LIN {X 0,Y 591.397,Z 324.376,A -85,B 0,C 180,E1 -9125.475,E2 -9125.475} C_VEL
LIN {X 0,Y 591.383,Z 324.375,A -85,B 0,C 180,E1 -9128.017,E2 -9128.017} C_VEL
LIN {X 0,Y 591.414,Z 324.373,A -85,B 0,C 180,E1 -9130.713,E2 -9130.713} C_VEL
LIN {X 0,Y 591.421,Z 324.373,A -85,B 0,C 180,E1 -9133.743,E2 -9133.743} C_VEL
LIN {X 0,Y 591.409,Z 324.376,A -85,B 0,C 180,E1 -9136.612,E2 -9136.612} C_VEL
LIN {X 0,Y 591.432,Z 324.373,A -85,B 0,C 180,E1 -9139.355,E2 -9139.355} C_VEL
LIN {X 0,Y 591.387,Z 324.373,A -85,B 0,C 180,E1 -9141.983,E2 -9141.983} C_VEL
LIN {X 0,Y 591.454,Z 324.372,A -85,B 0,C 180,E1 -9144.529,E2 -9144.529} C_VEL
LIN {X 0,Y 591.403,Z 324.379,A -85,B 0,C 180,E1 -9147.236,E2 -9147.236} C_VEL
LIN {X 0,Y 591.415,Z 324.382,A -85,B 0,C 180,E1 -9149.835,E2 -9149.835} C_VEL
LIN {X 0,Y 591.457,Z 324.484,A -85,B 0,C 180,E1 -9151.821,E2 -9151.821} C_VEL
LIN {X 0,Y 595.055,Z 338.646,A -85,B 0,C 180,E1 -9153.458,E2 -9153.458} C_VEL
LIN {X 0,Y 596.01,Z 344.054,A -85,B 0,C 180,E1 -9154.055,E2 -9154.055} C_VEL
LIN {X 0,Y 595.353,Z 369.323,A -85,B 0,C 180,E1 -9156.59,E2 -9156.59} C_VEL
LIN {X 0,Y 594.51,Z 396.234,A -85,B 0,C 180,E1 -9159.301,E2 -9159.301} C_VEL
LIN {X 0,Y 593.8,Z 422.727,A -85,B 0,C 180,E1 -9161.962,E2 -9161.962} C_VEL
LIN {X 0,Y 593.404,Z 439.816,A -85,B 0,C 180,E1 -9163.676,E2 -9163.676} C_VEL
LIN {X 0,Y 595.77,Z 457.22,A -85,B 0,C 180,E1 -9164.027,E2 -9164.027} C_VEL
LIN {X 0,Y 594.456,Z 560.115,A -85,B 0,C 180,E1 -9165.501,E2 -9165.501} C_VEL
LIN {X 0,Y 594.101,Z 582.366,A -85,B 0,C 180,E1 -9165.839,E2 -9165.839} C_VEL
LIN {X 0,Y 593.767,Z 596.032,A -85,B 0,C 180,E1 -9166.18,E2 -9166.18} C_VEL
LIN {X 0,Y 593.41,Z 609.595,A -85,B 0,C 180,E1 -9166.649,E2 -9166.649} C_VEL
LIN {X 0,Y 592.899,Z 623.687,A -85,B 0,C 180,E1 -9167.289,E2 -9167.289} C_VEL
LIN {X 0,Y 592.458,Z 635.61,A -85,B 0,C 180,E1 -9167.973,E2 -9167.973} C_VEL
LIN {X 0,Y 592.066,Z 646.637,A -85,B 0,C 180,E1 -9168.744,E2 -9168.744} C_VEL
LIN {X 0,Y 591.674,Z 657.474,A -85,B 0,C 180,E1 -9169.656,E2 -9169.656} C_VEL
LIN {X 0,Y 591.308,Z 667.035,A -85,B 0,C 180,E1 -9170.626,E2 -9170.626} C_VEL
LIN {X 0,Y 590.979,Z 675.465,A -85,B 0,C 180,E1 -9171.652,E2 -9171.652} C_VEL
LIN {X 0,Y 590.721,Z 683.499,A -85,B 0,C 180,E1 -9172.848,E2 -9172.848} C_VEL
LIN {X 0,Y 590.563,Z 689.147,A -85,B 0,C 180,E1 -9173.872,E2 -9173.872} C_VEL
LIN {X 0,Y 590.376,Z 695.034,A -85,B 0,C 180,E1 -9175.236,E2 -9175.236} C_VEL
LIN {X 0,Y 590.346,Z 699.319,A -85,B 0,C 180,E1 -9176.599,E2 -9176.599} C_VEL
LIN {X 0,Y 590.252,Z 702.124,A -85,B 0,C 180,E1 -9177.96,E2 -9177.96} C_VEL
LIN {X 0,Y 590.247,Z 703.522,A -85,B 0,C 180,E1 -9179.32,E2 -9179.32} C_VEL
LIN {X 0,Y 590.246,Z 703.516,A -85,B 0,C 180,E1 -9180.68,E2 -9180.68} C_VEL
LIN {X 0,Y 590.25,Z 702.107,A -85,B 0,C 180,E1 -9182.04,E2 -9182.04} C_VEL
LIN {X 0,Y 590.344,Z 699.294,A -85,B 0,C 180,E1 -9183.401,E2 -9183.401} C_VEL
LIN {X 0,Y 590.414,Z 695.001,A -85,B 0,C 180,E1 -9184.764,E2 -9184.764} C_VEL
LIN {X 0,Y 590.509,Z 689.102,A -85,B 0,C 180,E1 -9186.129,E2 -9186.129} C_VEL
LIN {X 0,Y 590.692,Z 682.418,A -85,B 0,C 180,E1 -9187.324,E2 -9187.324} C_VEL
LIN {X 0,Y 590.935,Z 674.066,A -85,B 0,C 180,E1 -9188.521,E2 -9188.521} C_VEL
LIN {X 0,Y 591.277,Z 665.351,A -85,B 0,C 180,E1 -9189.547,E2 -9189.547} C_VEL
LIN {X 0,Y 591.649,Z 654.979,A -85,B 0,C 180,E1 -9190.558,E2 -9190.558} C_VEL
LIN {X 0,Y 591.972,Z 644.168,A -85,B 0,C 180,E1 -9191.431,E2 -9191.431} C_VEL
LIN {X 0,Y 592.438,Z 632.612,A -85,B 0,C 180,E1 -9192.201,E2 -9192.201} C_VEL
LIN {X 0,Y 592.904,Z 619.997,A -85,B 0,C 180,E1 -9192.885,E2 -9192.885} C_VEL
LIN {X 0,Y 593.321,Z 607.005,A -85,B 0,C 180,E1 -9193.44,E2 -9193.44} C_VEL
LIN {X 0,Y 593.593,Z 593.037,A -85,B 0,C 180,E1 -9193.89,E2 -9193.89} C_VEL
LIN {X 0,Y 593.869,Z 578.644,A -85,B 0,C 180,E1 -9194.21,E2 -9194.21} C_VEL
LIN {X 0,Y 595.053,Z 455.793,A -85,B 0,C 180,E1 -9195.884,E2 -9195.884} C_VEL
LIN {X 0,Y 592.977,Z 439.459,A -85,B 0,C 180,E1 -9196.183,E2 -9196.183} C_VEL
LIN {X 0,Y 593.75,Z 410.791,A -85,B 0,C 180,E1 -9199.109,E2 -9199.109} C_VEL
LIN {X 0,Y 594.617,Z 381.153,A -85,B 0,C 180,E1 -9202.145,E2 -9202.145} C_VEL
LIN {X 0,Y 595.362,Z 356.403,A -85,B 0,C 180,E1 -9204.687,E2 -9204.687} C_VEL
LIN {X 0,Y 595.7,Z 344.018,A -85,B 0,C 180,E1 -9205.968,E2 -9205.968} C_VEL
LIN {X 0,Y 592.914,Z 330.893,A -85,B 0,C 180,E1 -9207.435,E2 -9207.435} C_VEL
LIN {X 0,Y 591.482,Z 324.367,A -85,B 0,C 180,E1 -9208.178,E2 -9208.178} C_VEL
LIN {X 0,Y 591.442,Z 324.368,A -85,B 0,C 180,E1 -9210.614,E2 -9210.614} C_VEL
LIN {X 0,Y 591.441,Z 324.372,A -85,B 0,C 180,E1 -9213.01,E2 -9213.01} C_VEL
LIN {X 0,Y 591.491,Z 324.365,A -85,B 0,C 180,E1 -9215.469,E2 -9215.469} C_VEL
LIN {X 0,Y 591.422,Z 324.368,A -85,B 0,C 180,E1 -9218.015,E2 -9218.015} C_VEL
LIN {X 0,Y 591.449,Z 324.368,A -85,B 0,C 180,E1 -9220.717,E2 -9220.717} C_VEL
LIN {X 0,Y 591.424,Z 324.371,A -85,B 0,C 180,E1 -9223.387,E2 -9223.387} C_VEL
LIN {X 0,Y 591.435,Z 324.367,A -85,B 0,C 180,E1 -9226.256,E2 -9226.256} C_VEL
LIN {X 0,Y 591.439,Z 324.37,A -85,B 0,C 180,E1 -9228.455,E2 -9228.455} C_VEL
LIN {X 0,Y 591.415,Z 324.372,A -85,B 0,C 180,E1 -9231.119,E2 -9231.119} C_VEL
LIN {X 0,Y 591.426,Z 324.37,A -85,B 0,C 180,E1 -9232.22,E2 -9232.22} C_VEL
LIN {X 0,Y 590.787,Z 324.455,A -85,B 0,C 180,E1 -9232.788,E2 -9232.788} C_VEL
LIN {X 0,Y 587.96,Z 324.808,A -85,B 0,C 180,E1 -9233.711,E2 -9233.711} C_VEL
LIN {X 0,Y 585.55,Z 325.106,A -85,B 0,C 180,E1 -9234.454,E2 -9234.454} C_VEL
LIN {X 0,Y 584.503,Z 325.233,A -85,B 0,C 180,E1 -9235.027,E2 -9235.027} C_VEL
LIN {X 0,Y 584.412,Z 325.242,A -85,B 0,C 180,E1 -9235.221,E2 -9235.221} C_VEL
LIN {X 0,Y 584.395,Z 325.248,A -85,B 0,C 180,E1 -9238.172,E2 -9238.172} C_VEL
LIN {X 0,Y 584.426,Z 325.241,A -85,B 0,C 180,E1 -9241.036,E2 -9241.036} C_VEL
LIN {X 0,Y 584.36,Z 325.249,A -85,B 0,C 180,E1 -9243.673,E2 -9243.673} C_VEL
LIN {X 0,Y 584.413,Z 325.246,A -85,B 0,C 180,E1 -9245.952,E2 -9245.952} C_VEL
LIN {X 0,Y 584.451,Z 325.237,A -85,B 0,C 180,E1 -9248.928,E2 -9248.928} C_VEL
LIN {X 0,Y 584.403,Z 325.249,A -85,B 0,C 180,E1 -9251.843,E2 -9251.843} C_VEL
LIN {X 0,Y 584.433,Z 325.24,A -85,B 0,C 180,E1 -9254.712,E2 -9254.712} C_VEL
LIN {X 0,Y 584.455,Z 325.237,A -85,B 0,C 180,E1 -9256.838,E2 -9256.838} C_VEL
LIN {X 0,Y 584.458,Z 325.239,A -85,B 0,C 180,E1 -9258.945,E2 -9258.945} C_VEL
LIN {X 0,Y 588.396,Z 337.126,A -85,B 0,C 180,E1 -9259.205,E2 -9259.205} C_VEL
LIN {X 0,Y 587.901,Z 445.913,A -85,B 0,C 180,E1 -9260.55,E2 -9260.55} C_VEL
LIN {X 0,Y 587.79,Z 460.378,A -85,B 0,C 180,E1 -9260.851,E2 -9260.851} C_VEL
LIN {X 0,Y 587.602,Z 473.525,A -85,B 0,C 180,E1 -9261.258,E2 -9261.258} C_VEL
LIN {X 0,Y 587.302,Z 485.998,A -85,B 0,C 180,E1 -9261.772,E2 -9261.772} C_VEL
LIN {X 0,Y 586.938,Z 498.954,A -85,B 0,C 180,E1 -9262.457,E2 -9262.457} C_VEL
LIN {X 0,Y 586.539,Z 510.662,A -85,B 0,C 180,E1 -9263.228,E2 -9263.228} C_VEL
LIN {X 0,Y 586.082,Z 520.417,A -85,B 0,C 180,E1 -9263.997,E2 -9263.997} C_VEL
LIN {X 0,Y 585.592,Z 531.141,A -85,B 0,C 180,E1 -9265.025,E2 -9265.025} C_VEL
LIN {X 0,Y 585.201,Z 540,A -85,B 0,C 180,E1 -9266.054,E2 -9266.054} C_VEL
LIN {X 0,Y 584.818,Z 548.476,A -85,B 0,C 180,E1 -9267.254,E2 -9267.254} C_VEL
LIN {X 0,Y 584.51,Z 554.451,A -85,B 0,C 180,E1 -9268.283,E2 -9268.283} C_VEL
LIN {X 0,Y 584.27,Z 559.407,A -85,B 0,C 180,E1 -9269.313,E2 -9269.313} C_VEL
LIN {X 0,Y 583.986,Z 564.529,A -85,B 0,C 180,E1 -9270.687,E2 -9270.687} C_VEL
LIN {X 0,Y 583.898,Z 568.164,A -85,B 0,C 180,E1 -9272.063,E2 -9272.063} C_VEL
LIN {X 0,Y 583.945,Z 570.435,A -85,B 0,C 180,E1 -9273.439,E2 -9273.439} C_VEL
LIN {X 0,Y 583.832,Z 571.428,A -85,B 0,C 180,E1 -9274.818,E2 -9274.818} C_VEL
LIN {X 0,Y 583.931,Z 571.112,A -85,B 0,C 180,E1 -9276.198,E2 -9276.198} C_VEL
LIN {X 0,Y 584.001,Z 569.505,A -85,B 0,C 180,E1 -9277.581,E2 -9277.581} C_VEL
LIN {X 0,Y 584.104,Z 566.555,A -85,B 0,C 180,E1 -9278.969,E2 -9278.969} C_VEL
LIN {X 0,Y 584.448,Z 562.149,A -85,B 0,C 180,E1 -9280.357,E2 -9280.357} C_VEL
LIN {X 0,Y 584.647,Z 557.768,A -85,B 0,C 180,E1 -9281.402,E2 -9281.402} C_VEL
LIN {X 0,Y 584.964,Z 552.416,A -85,B 0,C 180,E1 -9282.447,E2 -9282.447} C_VEL
LIN {X 0,Y 585.399,Z 544.728,A -85,B 0,C 180,E1 -9283.669,E2 -9283.669} C_VEL
LIN {X 0,Y 585.867,Z 536.664,A -85,B 0,C 180,E1 -9284.718,E2 -9284.718} C_VEL
LIN {X 0,Y 586.358,Z 526.909,A -85,B 0,C 180,E1 -9285.769,E2 -9285.769} C_VEL
LIN {X 0,Y 586.796,Z 517.087,A -85,B 0,C 180,E1 -9286.648,E2 -9286.648} C_VEL
LIN {X 0,Y 587.203,Z 506.593,A -85,B 0,C 180,E1 -9287.431,E2 -9287.431} C_VEL
LIN {X 0,Y 587.739,Z 494.971,A -85,B 0,C 180,E1 -9288.141,E2 -9288.141} C_VEL
LIN {X 0,Y 588.097,Z 482.425,A -85,B 0,C 180,E1 -9288.759,E2 -9288.759} C_VEL
LIN {X 0,Y 588.319,Z 469.674,A -85,B 0,C 180,E1 -9289.247,E2 -9289.247} C_VEL
LIN {X 0,Y 588.494,Z 455.956,A -85,B 0,C 180,E1 -9289.631,E2 -9289.631} C_VEL
LIN {X 0,Y 588.639,Z 442.281,A -85,B 0,C 180,E1 -9289.877,E2 -9289.877} C_VEL
LIN {X 0,Y 589.266,Z 338.454,A -85,B 0,C 180,E1 -9291.162,E2 -9291.162} C_VEL
LIN {X 0,Y 584.397,Z 325.318,A -85,B 0,C 180,E1 -9291.488,E2 -9291.488} C_VEL
LIN {X 0,Y 584.399,Z 325.253,A -85,B 0,C 180,E1 -9294.367,E2 -9294.367} C_VEL
LIN {X 0,Y 584.392,Z 325.248,A -85,B 0,C 180,E1 -9297.506,E2 -9297.506} C_VEL
LIN {X 0,Y 584.358,Z 325.257,A -85,B 0,C 180,E1 -9300.341,E2 -9300.341} C_VEL
LIN {X 0,Y 584.359,Z 325.25,A -85,B 0,C 180,E1 -9302.959,E2 -9302.959} C_VEL
LIN {X 0,Y 584.365,Z 325.253,A -85,B 0,C 180,E1 -9305.968,E2 -9305.968} C_VEL
LIN {X 0,Y 584.364,Z 325.249,A -85,B 0,C 180,E1 -9308.819,E2 -9308.819} C_VEL
LIN {X 0,Y 584.345,Z 325.251,A -85,B 0,C 180,E1 -9311.245,E2 -9311.245} C_VEL
LIN {X 0,Y 584.397,Z 325.252,A -85,B 0,C 180,E1 -9314.042,E2 -9314.042} C_VEL
LIN {X 0,Y 584.394,Z 325.244,A -85,B 0,C 180,E1 -9316.982,E2 -9316.982} C_VEL
LIN {X 0,Y 584.359,Z 325.253,A -85,B 0,C 180,E1 -9320.098,E2 -9320.098} C_VEL
LIN {X 0,Y 584.342,Z 325.238,A -85,B 0,C 180,E1 -9322.314,E2 -9322.314} C_VEL
LIN {X 0,Y 584.353,Z 325.24,A -85,B 0,C 180,E1 -9324.875,E2 -9324.875} C_VEL
LIN {X 0,Y 584.358,Z 325.249,A -85,B 0,C 180,E1 -9327.357,E2 -9327.357} C_VEL
LIN {X 0,Y 584.371,Z 325.248,A -85,B 0,C 180,E1 -9329.773,E2 -9329.773} C_VEL
LIN {X 0,Y 584.392,Z 325.242,A -85,B 0,C 180,E1 -9332.494,E2 -9332.494} C_VEL
LIN {X 0,Y 584.399,Z 325.248,A -85,B 0,C 180,E1 -9335.633,E2 -9335.633} C_VEL
LIN {X 0,Y 584.372,Z 325.244,A -85,B 0,C 180,E1 -9338.187,E2 -9338.187} C_VEL
LIN {X 0,Y 584.372,Z 325.25,A -85,B 0,C 180,E1 -9340.39,E2 -9340.39} C_VEL
LIN {X 0,Y 584.408,Z 325.251,A -85,B 0,C 180,E1 -9343.08,E2 -9343.08} C_VEL
LIN {X 0,Y 588.095,Z 337.425,A -85,B 0,C 180,E1 -9343.346,E2 -9343.346} C_VEL
LIN {X 0,Y 587.069,Z 446.386,A -85,B 0,C 180,E1 -9344.858,E2 -9344.858} C_VEL
LIN {X 0,Y 586.891,Z 461.083,A -85,B 0,C 180,E1 -9345.208,E2 -9345.208} C_VEL
LIN {X 0,Y 586.707,Z 475.547,A -85,B 0,C 180,E1 -9345.701,E2 -9345.701} C_VEL
LIN {X 0,Y 586.399,Z 488.186,A -85,B 0,C 180,E1 -9346.266,E2 -9346.266} C_VEL
LIN {X 0,Y 586.061,Z 500.538,A -85,B 0,C 180,E1 -9346.962,E2 -9346.962} C_VEL
LIN {X 0,Y 585.664,Z 512.992,A -85,B 0,C 180,E1 -9347.831,E2 -9347.831} C_VEL
LIN {X 0,Y 585.28,Z 524.558,A -85,B 0,C 180,E1 -9348.819,E2 -9348.819} C_VEL
LIN {X 0,Y 585.02,Z 534.267,A -85,B 0,C 180,E1 -9349.828,E2 -9349.828} C_VEL
LIN {X 0,Y 584.669,Z 542.575,A -85,B 0,C 180,E1 -9350.866,E2 -9350.866} C_VEL
LIN {X 0,Y 584.376,Z 550.49,A -85,B 0,C 180,E1 -9352.077,E2 -9352.077} C_VEL
LIN {X 0,Y 584.167,Z 556.045,A -85,B 0,C 180,E1 -9353.113,E2 -9353.113} C_VEL
LIN {X 0,Y 583.969,Z 561.848,A -85,B 0,C 180,E1 -9354.493,E2 -9354.493} C_VEL
LIN {X 0,Y 583.887,Z 566.071,A -85,B 0,C 180,E1 -9355.872,E2 -9355.872} C_VEL
LIN {X 0,Y 583.89,Z 568.829,A -85,B 0,C 180,E1 -9357.249,E2 -9357.249} C_VEL
LIN {X 0,Y 583.722,Z 570.182,A -85,B 0,C 180,E1 -9358.625,E2 -9358.625} C_VEL
LIN {X 0,Y 583.655,Z 570.168,A -85,B 0,C 180,E1 -9360,E2 -9360} C_VEL
LIN {X 0,Y 583.751,Z 568.777,A -85,B 0,C 180,E1 -9361.375,E2 -9361.375} C_VEL
LIN {X 0,Y 584.059,Z 565.978,A -85,B 0,C 180,E1 -9362.749,E2 -9362.749} C_VEL
LIN {X 0,Y 584.433,Z 561.687,A -85,B 0,C 180,E1 -9364.124,E2 -9364.124} C_VEL
LIN {X 0,Y 584.407,Z 555.792,A -85,B 0,C 180,E1 -9365.502,E2 -9365.502} C_VEL
LIN {X 0,Y 584.916,Z 549.091,A -85,B 0,C 180,E1 -9366.705,E2 -9366.705} C_VEL
LIN {X 0,Y 585.301,Z 540.781,A -85,B 0,C 180,E1 -9367.91,E2 -9367.91} C_VEL
LIN {X 0,Y 585.641,Z 532.032,A -85,B 0,C 180,E1 -9368.945,E2 -9368.945} C_VEL
LIN {X 0,Y 586.047,Z 521.342,A -85,B 0,C 180,E1 -9369.98,E2 -9369.98} C_VEL
LIN {X 0,Y 586.402,Z 512.877,A -85,B 0,C 180,E1 -9370.669,E2 -9370.669} C_VEL
LIN {X 0,Y 586.82,Z 501.498,A -85,B 0,C 180,E1 -9371.446,E2 -9371.446} C_VEL
LIN {X 0,Y 587.254,Z 488.639,A -85,B 0,C 180,E1 -9372.154,E2 -9372.154} C_VEL
LIN {X 0,Y 587.518,Z 475.083,A -85,B 0,C 180,E1 -9372.742,E2 -9372.742} C_VEL
LIN {X 0,Y 587.697,Z 460.944,A -85,B 0,C 180,E1 -9373.198,E2 -9373.198} C_VEL
LIN {X 0,Y 587.824,Z 446.981,A -85,B 0,C 180,E1 -9373.502,E2 -9373.502} C_VEL
LIN {X 0,Y 589.193,Z 337.801,A -85,B 0,C 180,E1 -9375.112,E2 -9375.112} C_VEL
LIN {X 0,Y 584.475,Z 325.436,A -85,B 0,C 180,E1 -9375.495,E2 -9375.495} C_VEL
LIN {X 0,Y 584.403,Z 325.252,A -85,B 0,C 180,E1 -9378.157,E2 -9378.157} C_VEL
LIN {X 0,Y 584.45,Z 325.241,A -85,B 0,C 180,E1 -9381.072,E2 -9381.072} C_VEL
LIN {X 0,Y 584.432,Z 325.249,A -85,B 0,C 180,E1 -9384.047,E2 -9384.047} C_VEL
LIN {X 0,Y 584.375,Z 325.25,A -85,B 0,C 180,E1 -9387.095,E2 -9387.095} C_VEL
LIN {X 0,Y 584.406,Z 325.247,A -85,B 0,C 180,E1 -9389.433,E2 -9389.433} C_VEL
LIN {X 0,Y 584.395,Z 325.249,A -85,B 0,C 180,E1 -9391.828,E2 -9391.828} C_VEL
LIN {X 0,Y 584.405,Z 325.242,A -85,B 0,C 180,E1 -9394.286,E2 -9394.286} C_VEL
LIN {X 0,Y 584.423,Z 325.239,A -85,B 0,C 180,E1 -9396.817,E2 -9396.817} C_VEL
LIN {X 0,Y 584.359,Z 325.246,A -85,B 0,C 180,E1 -9399.902,E2 -9399.902} C_VEL
LIN {X 0,Y 584.393,Z 325.24,A -85,B 0,C 180,E1 -9402.16,E2 -9402.16} C_VEL
LIN {X 0,Y 584.394,Z 325.249,A -85,B 0,C 180,E1 -9405.005,E2 -9405.005} C_VEL
LIN {X 0,Y 584.388,Z 325.244,A -85,B 0,C 180,E1 -9407.999,E2 -9407.999} C_VEL
LIN {X 0,Y 584.352,Z 325.254,A -85,B 0,C 180,E1 -9410.558,E2 -9410.558} C_VEL
LIN {X 0,Y 584.359,Z 325.251,A -85,B 0,C 180,E1 -9413.427,E2 -9413.427} C_VEL
LIN {X 0,Y 584.331,Z 325.249,A -85,B 0,C 180,E1 -9415.803,E2 -9415.803} C_VEL
LIN {X 0,Y 584.383,Z 325.253,A -85,B 0,C 180,E1 -9418.322,E2 -9418.322} C_VEL
LIN {X 0,Y 584.394,Z 325.249,A -85,B 0,C 180,E1 -9421.351,E2 -9421.351} C_VEL
LIN {X 0,Y 584.426,Z 325.373,A -85,B 0,C 180,E1 -9421.646,E2 -9421.646} C_VEL
LIN {X 0,Y 588.255,Z 343.449,A -85,B 0,C 180,E1 -9423.86,E2 -9423.86} C_VEL
LIN {X 0,Y 587.403,Z 365.293,A -85,B 0,C 180,E1 -9426.266,E2 -9426.266} C_VEL
LIN {X 0,Y 586.297,Z 393.805,A -85,B 0,C 180,E1 -9429.364,E2 -9429.364} C_VEL
LIN {X 0,Y 585.464,Z 418.853,A -85,B 0,C 180,E1 -9432.057,E2 -9432.057} C_VEL
LIN {X 0,Y 585.077,Z 431.768,A -85,B 0,C 180,E1 -9433.438,E2 -9433.438} C_VEL
LIN {X 0,Y 588.218,Z 459.236,A -85,B 0,C 180,E1 -9433.885,E2 -9433.885} C_VEL
LIN {X 0,Y 588.563,Z 466.079,A -85,B 0,C 180,E1 -9433.981,E2 -9433.981} C_VEL
LIN {X 0,Y 587.657,Z 571.482,A -85,B 0,C 180,E1 -9435.287,E2 -9435.287} C_VEL
LIN {X 0,Y 587.212,Z 585.956,A -85,B 0,C 180,E1 -9435.603,E2 -9435.603} C_VEL
LIN {X 0,Y 586.633,Z 599.953,A -85,B 0,C 180,E1 -9436.052,E2 -9436.052} C_VEL
LIN {X 0,Y 586.09,Z 613.003,A -85,B 0,C 180,E1 -9436.611,E2 -9436.611} C_VEL
LIN {X 0,Y 585.491,Z 625.675,A -85,B 0,C 180,E1 -9437.301,E2 -9437.301} C_VEL
LIN {X 0,Y 584.924,Z 641.523,A -85,B 0,C 180,E1 -9438.254,E2 -9438.254} C_VEL
LIN {X 0,Y 584.541,Z 653.444,A -85,B 0,C 180,E1 -9439.136,E2 -9439.136} C_VEL
LIN {X 0,Y 584.21,Z 662.96,A -85,B 0,C 180,E1 -9439.988,E2 -9439.988} C_VEL
LIN {X 0,Y 583.917,Z 672.662,A -85,B 0,C 180,E1 -9441.028,E2 -9441.028} C_VEL
LIN {X 0,Y 583.658,Z 681.865,A -85,B 0,C 180,E1 -9442.241,E2 -9442.241} C_VEL
LIN {X 0,Y 583.481,Z 689.238,A -85,B 0,C 180,E1 -9443.451,E2 -9443.451} C_VEL
LIN {X 0,Y 583.422,Z 694.371,A -85,B 0,C 180,E1 -9444.488,E2 -9444.488} C_VEL
LIN {X 0,Y 583.291,Z 699.616,A -85,B 0,C 180,E1 -9445.868,E2 -9445.868} C_VEL
LIN {X 0,Y 583.27,Z 703.288,A -85,B 0,C 180,E1 -9447.247,E2 -9447.247} C_VEL
LIN {X 0,Y 583.251,Z 705.492,A -85,B 0,C 180,E1 -9448.624,E2 -9448.624} C_VEL
LIN {X 0,Y 583.252,Z 706.28,A -85,B 0,C 180,E1 -9450,E2 -9450} C_VEL
LIN {X 0,Y 583.25,Z 705.646,A -85,B 0,C 180,E1 -9451.376,E2 -9451.376} C_VEL
LIN {X 0,Y 583.27,Z 703.57,A -85,B 0,C 180,E1 -9452.753,E2 -9452.753} C_VEL
LIN {X 0,Y 583.308,Z 700.026,A -85,B 0,C 180,E1 -9454.132,E2 -9454.132} C_VEL
LIN {X 0,Y 583.422,Z 694.91,A -85,B 0,C 180,E1 -9455.511,E2 -9455.511} C_VEL
LIN {X 0,Y 583.501,Z 689.927,A -85,B 0,C 180,E1 -9456.548,E2 -9456.548} C_VEL
LIN {X 0,Y 583.682,Z 682.734,A -85,B 0,C 180,E1 -9457.759,E2 -9457.759} C_VEL
LIN {X 0,Y 583.902,Z 675.173,A -85,B 0,C 180,E1 -9458.798,E2 -9458.798} C_VEL
LIN {X 0,Y 584.258,Z 666.053,A -85,B 0,C 180,E1 -9459.836,E2 -9459.836} C_VEL
LIN {X 0,Y 584.613,Z 656.484,A -85,B 0,C 180,E1 -9460.744,E2 -9460.744} C_VEL
LIN {X 0,Y 585.045,Z 644.9,A -85,B 0,C 180,E1 -9461.656,E2 -9461.656} C_VEL
LIN {X 0,Y 585.416,Z 632.766,A -85,B 0,C 180,E1 -9462.437,E2 -9462.437} C_VEL
LIN {X 0,Y 585.937,Z 619.165,A -85,B 0,C 180,E1 -9463.128,E2 -9463.128} C_VEL
LIN {X 0,Y 586.311,Z 604.779,A -85,B 0,C 180,E1 -9463.691,E2 -9463.691} C_VEL
LIN {X 0,Y 586.943,Z 582.569,A -85,B 0,C 180,E1 -9464.315,E2 -9464.315} C_VEL
LIN {X 0,Y 587.347,Z 568.106,A -85,B 0,C 180,E1 -9464.59,E2 -9464.59} C_VEL
LIN {X 0,Y 587.831,Z 505.932,A -85,B 0,C 180,E1 -9465.374,E2 -9465.374} C_VEL
LIN {X 0,Y 588.355,Z 461.363,A -85,B 0,C 180,E1 -9466.058,E2 -9466.058} C_VEL
LIN {X 0,Y 586.017,Z 437.005,A -85,B 0,C 180,E1 -9466.538,E2 -9466.538} C_VEL
LIN {X 0,Y 585.044,Z 427.965,A -85,B 0,C 180,E1 -9466.779,E2 -9466.779} C_VEL
LIN {X 0,Y 585.853,Z 398.261,A -85,B 0,C 180,E1 -9469.922,E2 -9469.922} C_VEL
LIN {X 0,Y 586.666,Z 372.688,A -85,B 0,C 180,E1 -9472.647,E2 -9472.647} C_VEL
LIN {X 0,Y 587.629,Z 345.22,A -85,B 0,C 180,E1 -9475.601,E2 -9475.601} C_VEL
LIN {X 0,Y 587.678,Z 341.765,A -85,B 0,C 180,E1 -9475.977,E2 -9475.977} C_VEL
LIN {X 0,Y 584.405,Z 325.25,A -85,B 0,C 180,E1 -9477.917,E2 -9477.917} C_VEL
LIN {X 0,Y 584.354,Z 325.25,A -85,B 0,C 180,E1 -9480.341,E2 -9480.341} C_VEL
LIN {X 0,Y 584.357,Z 325.251,A -85,B 0,C 180,E1 -9482.959,E2 -9482.959} C_VEL
LIN {X 0,Y 584.346,Z 325.253,A -85,B 0,C 180,E1 -9485.97,E2 -9485.97} C_VEL
LIN {X 0,Y 584.349,Z 325.253,A -85,B 0,C 180,E1 -9488.818,E2 -9488.818} C_VEL
LIN {X 0,Y 584.34,Z 325.254,A -85,B 0,C 180,E1 -9491.245,E2 -9491.245} C_VEL
LIN {X 0,Y 584.392,Z 325.247,A -85,B 0,C 180,E1 -9494.042,E2 -9494.042} C_VEL
LIN {X 0,Y 584.357,Z 325.253,A -85,B 0,C 180,E1 -9496.986,E2 -9496.986} C_VEL
LIN {X 0,Y 584.355,Z 325.251,A -85,B 0,C 180,E1 -9500.098,E2 -9500.098} C_VEL
LIN {X 0,Y 584.371,Z 325.249,A -85,B 0,C 180,E1 -9502.316,E2 -9502.316} C_VEL
LIN {X 0,Y 584.404,Z 325.249,A -85,B 0,C 180,E1 -9504.879,E2 -9504.879} C_VEL
LIN {X 0,Y 584.357,Z 325.258,A -85,B 0,C 180,E1 -9507.358,E2 -9507.358} C_VEL
LIN {X 0,Y 584.377,Z 325.259,A -85,B 0,C 180,E1 -9509.774,E2 -9509.774} C_VEL
LIN {X 0,Y 584.407,Z 325.27,A -85,B 0,C 180,E1 -9511.499,E2 -9511.499} C_VEL
LIN {X 0,Y 588.269,Z 340.159,A -85,B 0,C 180,E1 -9513.255,E2 -9513.255} C_VEL
LIN {X 0,Y 589.318,Z 345.96,A -85,B 0,C 180,E1 -9513.911,E2 -9513.911} C_VEL
LIN {X 0,Y 588.635,Z 370.358,A -85,B 0,C 180,E1 -9516.386,E2 -9516.386} C_VEL
LIN {X 0,Y 587.776,Z 396.637,A -85,B 0,C 180,E1 -9519.053,E2 -9519.053} C_VEL
LIN {X 0,Y 586.971,Z 423.126,A -85,B 0,C 180,E1 -9521.745,E2 -9521.745} C_VEL
LIN {X 0,Y 586.595,Z 439.961,A -85,B 0,C 180,E1 -9523.436,E2 -9523.436} C_VEL
LIN {X 0,Y 589.053,Z 457.646,A -85,B 0,C 180,E1 -9523.807,E2 -9523.807} C_VEL
LIN {X 0,Y 587.618,Z 560.787,A -85,B 0,C 180,E1 -9525.324,E2 -9525.324} C_VEL
LIN {X 0,Y 587.257,Z 581.978,A -85,B 0,C 180,E1 -9525.649,E2 -9525.649} C_VEL
LIN {X 0,Y 586.896,Z 596.435,A -85,B 0,C 180,E1 -9526.015,E2 -9526.015} C_VEL
LIN {X 0,Y 586.517,Z 609.87,A -85,B 0,C 180,E1 -9526.49,E2 -9526.49} C_VEL
LIN {X 0,Y 585.983,Z 623.876,A -85,B 0,C 180,E1 -9527.137,E2 -9527.137} C_VEL
LIN {X 0,Y 585.529,Z 635.745,A -85,B 0,C 180,E1 -9527.829,E2 -9527.829} C_VEL
LIN {X 0,Y 585.08,Z 646.743,A -85,B 0,C 180,E1 -9528.607,E2 -9528.607} C_VEL
LIN {X 0,Y 584.668,Z 657.182,A -85,B 0,C 180,E1 -9529.494,E2 -9529.494} C_VEL
LIN {X 0,Y 584.299,Z 667.131,A -85,B 0,C 180,E1 -9530.513,E2 -9530.513} C_VEL
LIN {X 0,Y 583.94,Z 675.544,A -85,B 0,C 180,E1 -9531.55,E2 -9531.55} C_VEL
LIN {X 0,Y 583.642,Z 683.568,A -85,B 0,C 180,E1 -9532.761,E2 -9532.761} C_VEL
LIN {X 0,Y 583.498,Z 689.205,A -85,B 0,C 180,E1 -9533.798,E2 -9533.798} C_VEL
LIN {X 0,Y 583.291,Z 695.093,A -85,B 0,C 180,E1 -9535.178,E2 -9535.178} C_VEL
LIN {X 0,Y 583.259,Z 699.374,A -85,B 0,C 180,E1 -9536.558,E2 -9536.558} C_VEL
LIN {X 0,Y 583.163,Z 702.17,A -85,B 0,C 180,E1 -9537.935,E2 -9537.935} C_VEL
LIN {X 0,Y 583.147,Z 703.55,A -85,B 0,C 180,E1 -9539.312,E2 -9539.312} C_VEL
LIN {X 0,Y 583.146,Z 703.517,A -85,B 0,C 180,E1 -9540.688,E2 -9540.688} C_VEL
LIN {X 0,Y 583.161,Z 702.083,A -85,B 0,C 180,E1 -9542.065,E2 -9542.065} C_VEL
LIN {X 0,Y 583.255,Z 699.239,A -85,B 0,C 180,E1 -9543.443,E2 -9543.443} C_VEL
LIN {X 0,Y 583.323,Z 694.911,A -85,B 0,C 180,E1 -9544.822,E2 -9544.822} C_VEL
LIN {X 0,Y 583.43,Z 688.966,A -85,B 0,C 180,E1 -9546.203,E2 -9546.203} C_VEL
LIN {X 0,Y 583.634,Z 682.22,A -85,B 0,C 180,E1 -9547.413,E2 -9547.413} C_VEL
LIN {X 0,Y 583.86,Z 673.804,A -85,B 0,C 180,E1 -9548.625,E2 -9548.625} C_VEL
LIN {X 0,Y 584.233,Z 665.021,A -85,B 0,C 180,E1 -9549.663,E2 -9549.663} C_VEL
LIN {X 0,Y 584.591,Z 655.602,A -85,B 0,C 180,E1 -9550.593,E2 -9550.593} C_VEL
LIN {X 0,Y 584.929,Z 644.812,A -85,B 0,C 180,E1 -9551.484,E2 -9551.484} C_VEL
LIN {X 0,Y 585.375,Z 633.371,A -85,B 0,C 180,E1 -9552.263,E2 -9552.263} C_VEL
LIN {X 0,Y 585.861,Z 620.916,A -85,B 0,C 180,E1 -9552.954,E2 -9552.954} C_VEL
LIN {X 0,Y 586.329,Z 607.105,A -85,B 0,C 180,E1 -9553.559,E2 -9553.559} C_VEL
LIN {X 0,Y 586.612,Z 593.187,A -85,B 0,C 180,E1 -9554.015,E2 -9554.015} C_VEL
LIN {X 0,Y 586.918,Z 578.92,A -85,B 0,C 180,E1 -9554.338,E2 -9554.338} C_VEL
LIN {X 0,Y 588.223,Z 456.806,A -85,B 0,C 180,E1 -9556.037,E2 -9556.037} C_VEL
LIN {X 0,Y 586.038,Z 439.461,A -85,B 0,C 180,E1 -9556.357,E2 -9556.357} C_VEL
LIN {X 0,Y 586.876,Z 409.273,A -85,B 0,C 180,E1 -9559.459,E2 -9559.459} C_VEL
LIN {X 0,Y 587.74,Z 380.6,A -85,B 0,C 180,E1 -9562.418,E2 -9562.418} C_VEL
LIN {X 0,Y 588.606,Z 354.291,A -85,B 0,C 180,E1 -9565.147,E2 -9565.147} C_VEL
LIN {X 0,Y 588.763,Z 344.951,A -85,B 0,C 180,E1 -9566.116,E2 -9566.116} C_VEL
LIN {X 0,Y 584.447,Z 325.243,A -85,B 0,C 180,E1 -9568.377,E2 -9568.377} C_VEL
LIN {X 0,Y 584.406,Z 325.248,A -85,B 0,C 180,E1 -9571.023,E2 -9571.023} C_VEL
LIN {X 0,Y 584.388,Z 325.251,A -85,B 0,C 180,E1 -9573.46,E2 -9573.46} C_VEL
LIN {X 0,Y 584.428,Z 325.239,A -85,B 0,C 180,E1 -9575.964,E2 -9575.964} C_VEL
LIN {X 0,Y 584.368,Z 325.251,A -85,B 0,C 180,E1 -9578.82,E2 -9578.82} C_VEL
LIN {X 0,Y 584.384,Z 325.25,A -85,B 0,C 180,E1 -9581.242,E2 -9581.242} C_VEL
LIN {X 0,Y 584.398,Z 325.243,A -85,B 0,C 180,E1 -9584.041,E2 -9584.041} C_VEL
LIN {X 0,Y 584.401,Z 325.25,A -85,B 0,C 180,E1 -9586.981,E2 -9586.981} C_VEL
LIN {X 0,Y 584.415,Z 325.241,A -85,B 0,C 180,E1 -9589.668,E2 -9589.668} C_VEL
LIN {X 0,Y 584.386,Z 325.248,A -85,B 0,C 180,E1 -9592.317,E2 -9592.317} C_VEL
LIN {X 0,Y 584.441,Z 325.242,A -85,B 0,C 180,E1 -9594.881,E2 -9594.881} C_VEL
LIN {X 0,Y 584.412,Z 325.242,A -85,B 0,C 180,E1 -9595.221,E2 -9595.221} C_VEL
LIN {X 0,Y 583.729,Z 325.327,A -85,B 0,C 180,E1 -9595.796,E2 -9595.796} C_VEL
LIN {X 0,Y 580.87,Z 325.688,A -85,B 0,C 180,E1 -9596.729,E2 -9596.729} C_VEL
LIN {X 0,Y 578.462,Z 325.986,A -85,B 0,C 180,E1 -9597.479,E2 -9597.479} C_VEL
LIN {X 0,Y 577.428,Z 326.115,A -85,B 0,C 180,E1 -9598.059,E2 -9598.059} C_VEL
LIN {X 0,Y 577.343,Z 326.126,A -85,B 0,C 180,E1 -9598.255,E2 -9598.255} C_VEL
LIN {X 0,Y 577.391,Z 326.117,A -85,B 0,C 180,E1 -9600.971,E2 -9600.971} C_VEL
LIN {X 0,Y 577.316,Z 326.128,A -85,B 0,C 180,E1 -9603.874,E2 -9603.874} C_VEL
LIN {X 0,Y 577.359,Z 326.126,A -85,B 0,C 180,E1 -9606.4,E2 -9606.4} C_VEL
LIN {X 0,Y 577.399,Z 326.116,A -85,B 0,C 180,E1 -9609.082,E2 -9609.082} C_VEL
LIN {X 0,Y 577.383,Z 326.12,A -85,B 0,C 180,E1 -9611.614,E2 -9611.614} C_VEL
LIN {X 0,Y 577.399,Z 326.117,A -85,B 0,C 180,E1 -9614.521,E2 -9614.521} C_VEL
LIN {X 0,Y 577.41,Z 326.114,A -85,B 0,C 180,E1 -9616.674,E2 -9616.674} C_VEL
LIN {X 0,Y 577.421,Z 326.115,A -85,B 0,C 180,E1 -9618.764,E2 -9618.764} C_VEL
LIN {X 0,Y 581.561,Z 338.528,A -85,B 0,C 180,E1 -9619.041,E2 -9619.041} C_VEL
LIN {X 0,Y 581.028,Z 446.658,A -85,B 0,C 180,E1 -9620.393,E2 -9620.393} C_VEL
LIN {X 0,Y 580.908,Z 461.132,A -85,B 0,C 180,E1 -9620.697,E2 -9620.697} C_VEL
LIN {X 0,Y 580.698,Z 474.286,A -85,B 0,C 180,E1 -9621.11,E2 -9621.11} C_VEL
LIN {X 0,Y 580.346,Z 487.65,A -85,B 0,C 180,E1 -9621.672,E2 -9621.672} C_VEL
LIN {X 0,Y 580.011,Z 500.411,A -85,B 0,C 180,E1 -9622.366,E2 -9622.366} C_VEL
LIN {X 0,Y 579.585,Z 511.999,A -85,B 0,C 180,E1 -9623.146,E2 -9623.146} C_VEL
LIN {X 0,Y 578.98,Z 523.573,A -85,B 0,C 180,E1 -9624.098,E2 -9624.098} C_VEL
LIN {X 0,Y 578.507,Z 533.897,A -85,B 0,C 180,E1 -9625.138,E2 -9625.138} C_VEL
LIN {X 0,Y 578.101,Z 542.423,A -85,B 0,C 180,E1 -9626.179,E2 -9626.179} C_VEL
LIN {X 0,Y 577.789,Z 550.598,A -85,B 0,C 180,E1 -9627.395,E2 -9627.395} C_VEL
LIN {X 0,Y 577.403,Z 557.205,A -85,B 0,C 180,E1 -9628.61,E2 -9628.61} C_VEL
LIN {X 0,Y 577.05,Z 563.084,A -85,B 0,C 180,E1 -9630,E2 -9630} C_VEL
LIN {X 0,Y 576.818,Z 567.406,A -85,B 0,C 180,E1 -9631.392,E2 -9631.392} C_VEL
LIN {X 0,Y 576.909,Z 570.295,A -85,B 0,C 180,E1 -9632.784,E2 -9632.784} C_VEL
LIN {X 0,Y 576.813,Z 571.892,A -85,B 0,C 180,E1 -9634.178,E2 -9634.178} C_VEL
LIN {X 0,Y 576.863,Z 572.185,A -85,B 0,C 180,E1 -9635.575,E2 -9635.575} C_VEL
LIN {X 0,Y 576.914,Z 571.193,A -85,B 0,C 180,E1 -9636.974,E2 -9636.974} C_VEL
LIN {X 0,Y 577.023,Z 568.882,A -85,B 0,C 180,E1 -9638.376,E2 -9638.376} C_VEL
LIN {X 0,Y 577.329,Z 565.172,A -85,B 0,C 180,E1 -9639.78,E2 -9639.78} C_VEL
LIN {X 0,Y 577.557,Z 559.926,A -85,B 0,C 180,E1 -9641.189,E2 -9641.189} C_VEL
LIN {X 0,Y 577.894,Z 554.878,A -85,B 0,C 180,E1 -9642.246,E2 -9642.246} C_VEL
LIN {X 0,Y 578.344,Z 547.617,A -85,B 0,C 180,E1 -9643.482,E2 -9643.482} C_VEL
LIN {X 0,Y 578.748,Z 540.45,A -85,B 0,C 180,E1 -9644.482,E2 -9644.482} C_VEL
LIN {X 0,Y 579.313,Z 530.768,A -85,B 0,C 180,E1 -9645.606,E2 -9645.606} C_VEL
LIN {X 0,Y 579.793,Z 520.521,A -85,B 0,C 180,E1 -9646.584,E2 -9646.584} C_VEL
LIN {X 0,Y 580.299,Z 509.298,A -85,B 0,C 180,E1 -9647.464,E2 -9647.464} C_VEL
LIN {X 0,Y 580.882,Z 496.54,A -85,B 0,C 180,E1 -9648.271,E2 -9648.271} C_VEL
LIN {X 0,Y 581.286,Z 484.205,A -85,B 0,C 180,E1 -9648.896,E2 -9648.896} C_VEL
LIN {X 0,Y 581.498,Z 473.078,A -85,B 0,C 180,E1 -9649.345,E2 -9649.345} C_VEL
LIN {X 0,Y 581.705,Z 459.207,A -85,B 0,C 180,E1 -9649.763,E2 -9649.763} C_VEL
LIN {X 0,Y 581.837,Z 444.96,A -85,B 0,C 180,E1 -9650.045,E2 -9650.045} C_VEL
LIN {X 0,Y 582.559,Z 340.091,A -85,B 0,C 180,E1 -9651.361,E2 -9651.361} C_VEL
LIN {X 0,Y 577.35,Z 326.13,A -85,B 0,C 180,E1 -9651.722,E2 -9651.722} C_VEL
LIN {X 0,Y 577.364,Z 326.13,A -85,B 0,C 180,E1 -9654.51,E2 -9654.51} C_VEL
LIN {X 0,Y 577.352,Z 326.126,A -85,B 0,C 180,E1 -9657.669,E2 -9657.669} C_VEL
LIN {X 0,Y 577.312,Z 326.133,A -85,B 0,C 180,E1 -9660.522,E2 -9660.522} C_VEL
LIN {X 0,Y 577.309,Z 326.127,A -85,B 0,C 180,E1 -9663.157,E2 -9663.157} C_VEL
LIN {X 0,Y 577.331,Z 326.126,A -85,B 0,C 180,E1 -9665.622,E2 -9665.622} C_VEL
LIN {X 0,Y 577.299,Z 326.136,A -85,B 0,C 180,E1 -9668.228,E2 -9668.228} C_VEL
LIN {X 0,Y 577.311,Z 326.128,A -85,B 0,C 180,E1 -9670.933,E2 -9670.933} C_VEL
LIN {X 0,Y 577.335,Z 326.129,A -85,B 0,C 180,E1 -9673.753,E2 -9673.753} C_VEL
LIN {X 0,Y 577.343,Z 326.129,A -85,B 0,C 180,E1 -9676.248,E2 -9676.248} C_VEL
LIN {X 0,Y 577.311,Z 326.125,A -85,B 0,C 180,E1 -9679.067,E2 -9679.067} C_VEL
LIN {X 0,Y 577.297,Z 326.125,A -85,B 0,C 180,E1 -9681.772,E2 -9681.772} C_VEL
LIN {X 0,Y 577.34,Z 326.116,A -85,B 0,C 180,E1 -9684.384,E2 -9684.384} C_VEL
LIN {X 0,Y 577.329,Z 326.122,A -85,B 0,C 180,E1 -9686.909,E2 -9686.909} C_VEL
LIN {X 0,Y 577.313,Z 326.125,A -85,B 0,C 180,E1 -9689.478,E2 -9689.478} C_VEL
LIN {X 0,Y 577.329,Z 326.131,A -85,B 0,C 180,E1 -9691.76,E2 -9691.76} C_VEL
LIN {X 0,Y 577.317,Z 326.125,A -85,B 0,C 180,E1 -9694.101,E2 -9694.101} C_VEL
LIN {X 0,Y 577.309,Z 326.127,A -85,B 0,C 180,E1 -9696.397,E2 -9696.397} C_VEL
LIN {X 0,Y 577.359,Z 326.121,A -85,B 0,C 180,E1 -9699.401,E2 -9699.401} C_VEL
LIN {X 0,Y 577.369,Z 326.132,A -85,B 0,C 180,E1 -9701.613,E2 -9701.613} C_VEL
LIN {X 0,Y 577.377,Z 326.126,A -85,B 0,C 180,E1 -9702.919,E2 -9702.919} C_VEL
LIN {X 0,Y 581.156,Z 338.121,A -85,B 0,C 180,E1 -9703.19,E2 -9703.19} C_VEL
LIN {X 0,Y 580.112,Z 447.095,A -85,B 0,C 180,E1 -9704.733,E2 -9704.733} C_VEL
LIN {X 0,Y 579.922,Z 462.081,A -85,B 0,C 180,E1 -9705.095,E2 -9705.095} C_VEL
LIN {X 0,Y 579.756,Z 475.829,A -85,B 0,C 180,E1 -9705.57,E2 -9705.57} C_VEL
LIN {X 0,Y 579.408,Z 489.433,A -85,B 0,C 180,E1 -9706.187,E2 -9706.187} C_VEL
LIN {X 0,Y 579.064,Z 501.679,A -85,B 0,C 180,E1 -9706.891,E2 -9706.891} C_VEL
LIN {X 0,Y 578.669,Z 514.075,A -85,B 0,C 180,E1 -9707.77,E2 -9707.77} C_VEL
LIN {X 0,Y 578.283,Z 524.298,A -85,B 0,C 180,E1 -9708.648,E2 -9708.648} C_VEL
LIN {X 0,Y 578.019,Z 534.491,A -85,B 0,C 180,E1 -9709.703,E2 -9709.703} C_VEL
LIN {X 0,Y 577.662,Z 542.913,A -85,B 0,C 180,E1 -9710.754,E2 -9710.754} C_VEL
LIN {X 0,Y 577.334,Z 550.931,A -85,B 0,C 180,E1 -9711.98,E2 -9711.98} C_VEL
LIN {X 0,Y 577.125,Z 556.561,A -85,B 0,C 180,E1 -9713.029,E2 -9713.029} C_VEL
LIN {X 0,Y 576.928,Z 562.433,A -85,B 0,C 180,E1 -9714.426,E2 -9714.426} C_VEL
LIN {X 0,Y 576.827,Z 566.726,A -85,B 0,C 180,E1 -9715.822,E2 -9715.822} C_VEL
LIN {X 0,Y 576.836,Z 569.547,A -85,B 0,C 180,E1 -9717.216,E2 -9717.216} C_VEL
LIN {X 0,Y 576.687,Z 570.96,A -85,B 0,C 180,E1 -9718.608,E2 -9718.608} C_VEL
LIN {X 0,Y 576.613,Z 570.993,A -85,B 0,C 180,E1 -9720,E2 -9720} C_VEL
LIN {X 0,Y 576.714,Z 569.643,A -85,B 0,C 180,E1 -9721.392,E2 -9721.392} C_VEL
LIN {X 0,Y 577.037,Z 566.883,A -85,B 0,C 180,E1 -9722.783,E2 -9722.783} C_VEL
LIN {X 0,Y 577.43,Z 562.646,A -85,B 0,C 180,E1 -9724.174,E2 -9724.174} C_VEL
LIN {X 0,Y 577.395,Z 558.428,A -85,B 0,C 180,E1 -9725.22,E2 -9725.22} C_VEL
LIN {X 0,Y 577.769,Z 553.16,A -85,B 0,C 180,E1 -9726.264,E2 -9726.264} C_VEL
LIN {X 0,Y 578.204,Z 545.616,A -85,B 0,C 180,E1 -9727.483,E2 -9727.483} C_VEL
LIN {X 0,Y 578.502,Z 537.709,A -85,B 0,C 180,E1 -9728.53,E2 -9728.53} C_VEL
LIN {X 0,Y 578.908,Z 528.123,A -85,B 0,C 180,E1 -9729.576,E2 -9729.576} C_VEL
LIN {X 0,Y 579.244,Z 517.44,A -85,B 0,C 180,E1 -9730.538,E2 -9730.538} C_VEL
LIN {X 0,Y 579.793,Z 506.832,A -85,B 0,C 180,E1 -9731.321,E2 -9731.321} C_VEL
LIN {X 0,Y 580.299,Z 494.761,A -85,B 0,C 180,E1 -9732.053,E2 -9732.053} C_VEL
LIN {X 0,Y 580.602,Z 481.089,A -85,B 0,C 180,E1 -9732.719,E2 -9732.719} C_VEL
LIN {X 0,Y 580.84,Z 467.325,A -85,B 0,C 180,E1 -9733.223,E2 -9733.223} C_VEL
LIN {X 0,Y 580.978,Z 452.999,A -85,B 0,C 180,E1 -9733.597,E2 -9733.597} C_VEL
LIN {X 0,Y 581.202,Z 426.55,A -85,B 0,C 180,E1 -9734.014,E2 -9734.014} C_VEL
LIN {X 0,Y 582.546,Z 339.393,A -85,B 0,C 180,E1 -9735.339,E2 -9735.339} C_VEL
LIN {X 0,Y 577.482,Z 326.603,A -85,B 0,C 180,E1 -9735.747,E2 -9735.747} C_VEL
LIN {X 0,Y 577.42,Z 326.121,A -85,B 0,C 180,E1 -9735.778,E2 -9735.778} C_VEL
LIN {X 0,Y 577.37,Z 326.124,A -85,B 0,C 180,E1 -9738.867,E2 -9738.867} C_VEL
LIN {X 0,Y 577.397,Z 326.12,A -85,B 0,C 180,E1 -9741.342,E2 -9741.342} C_VEL
LIN {X 0,Y 577.395,Z 326.122,A -85,B 0,C 180,E1 -9744.359,E2 -9744.359} C_VEL
LIN {X 0,Y 577.367,Z 326.126,A -85,B 0,C 180,E1 -9747.672,E2 -9747.672} C_VEL
LIN {X 0,Y 577.36,Z 326.127,A -85,B 0,C 180,E1 -9749.828,E2 -9749.828} C_VEL
LIN {X 0,Y 577.338,Z 326.125,A -85,B 0,C 180,E1 -9752.264,E2 -9752.264} C_VEL
LIN {X 0,Y 577.379,Z 326.117,A -85,B 0,C 180,E1 -9754.763,E2 -9754.763} C_VEL
LIN {X 0,Y 577.339,Z 326.124,A -85,B 0,C 180,E1 -9757.345,E2 -9757.345} C_VEL
LIN {X 0,Y 577.329,Z 326.12,A -85,B 0,C 180,E1 -9760.151,E2 -9760.151} C_VEL
LIN {X 0,Y 577.342,Z 326.122,A -85,B 0,C 180,E1 -9762.797,E2 -9762.797} C_VEL
LIN {X 0,Y 577.36,Z 326.119,A -85,B 0,C 180,E1 -9765.707,E2 -9765.707} C_VEL
LIN {X 0,Y 577.33,Z 326.123,A -85,B 0,C 180,E1 -9768.142,E2 -9768.142} C_VEL
LIN {X 0,Y 577.314,Z 326.132,A -85,B 0,C 180,E1 -9770.941,E2 -9770.941} C_VEL
LIN {X 0,Y 577.31,Z 326.128,A -85,B 0,C 180,E1 -9773.522,E2 -9773.522} C_VEL
LIN {X 0,Y 577.288,Z 326.128,A -85,B 0,C 180,E1 -9776.073,E2 -9776.073} C_VEL
LIN {X 0,Y 577.318,Z 326.133,A -85,B 0,C 180,E1 -9778.553,E2 -9778.553} C_VEL
LIN {X 0,Y 577.369,Z 326.253,A -85,B 0,C 180,E1 -9781.441,E2 -9781.441} C_VEL
LIN {X 0,Y 581.024,Z 342.828,A -85,B 0,C 180,E1 -9783.509,E2 -9783.509} C_VEL
LIN {X 0,Y 581.348,Z 346.234,A -85,B 0,C 180,E1 -9783.91,E2 -9783.91} C_VEL
LIN {X 0,Y 580.479,Z 366.4,A -85,B 0,C 180,E1 -9786.157,E2 -9786.157} C_VEL
LIN {X 0,Y 579.383,Z 393.2,A -85,B 0,C 180,E1 -9789.106,E2 -9789.106} C_VEL
LIN {X 0,Y 578.506,Z 416.566,A -85,B 0,C 180,E1 -9791.651,E2 -9791.651} C_VEL
LIN {X 0,Y 578.146,Z 431.018,A -85,B 0,C 180,E1 -9793.219,E2 -9793.219} C_VEL
LIN {X 0,Y 581.741,Z 462.875,A -85,B 0,C 180,E1 -9793.739,E2 -9793.739} C_VEL
LIN {X 0,Y 580.83,Z 570.776,A -85,B 0,C 180,E1 -9795.093,E2 -9795.093} C_VEL
LIN {X 0,Y 580.358,Z 585.032,A -85,B 0,C 180,E1 -9795.407,E2 -9795.407} C_VEL
LIN {X 0,Y 579.797,Z 598.498,A -85,B 0,C 180,E1 -9795.839,E2 -9795.839} C_VEL
LIN {X 0,Y 579.215,Z 610.803,A -85,B 0,C 180,E1 -9796.36,E2 -9796.36} C_VEL
LIN {X 0,Y 578.622,Z 623.745,A -85,B 0,C 180,E1 -9797.059,E2 -9797.059} C_VEL
LIN {X 0,Y 577.885,Z 642.195,A -85,B 0,C 180,E1 -9798.197,E2 -9798.197} C_VEL
LIN {X 0,Y 577.533,Z 652.476,A -85,B 0,C 180,E1 -9798.966,E2 -9798.966} C_VEL
LIN {X 0,Y 577.204,Z 662.531,A -85,B 0,C 180,E1 -9799.865,E2 -9799.865} C_VEL
LIN {X 0,Y 576.869,Z 672.308,A -85,B 0,C 180,E1 -9800.918,E2 -9800.918} C_VEL
LIN {X 0,Y 576.622,Z 680.381,A -85,B 0,C 180,E1 -9801.97,E2 -9801.97} C_VEL
LIN {X 0,Y 576.429,Z 687.064,A -85,B 0,C 180,E1 -9803.02,E2 -9803.02} C_VEL
LIN {X 0,Y 576.349,Z 692.575,A -85,B 0,C 180,E1 -9804.071,E2 -9804.071} C_VEL
LIN {X 0,Y 576.214,Z 698.115,A -85,B 0,C 180,E1 -9805.408,E2 -9805.408} C_VEL
LIN {X 0,Y 576.229,Z 701.544,A -85,B 0,C 180,E1 -9806.515,E2 -9806.515} C_VEL
LIN {X 0,Y 576.145,Z 704.507,A -85,B 0,C 180,E1 -9807.91,E2 -9807.91} C_VEL
LIN {X 0,Y 576.14,Z 706.029,A -85,B 0,C 180,E1 -9809.303,E2 -9809.303} C_VEL
LIN {X 0,Y 576.139,Z 706.134,A -85,B 0,C 180,E1 -9810.696,E2 -9810.696} C_VEL
LIN {X 0,Y 576.146,Z 704.802,A -85,B 0,C 180,E1 -9812.09,E2 -9812.09} C_VEL
LIN {X 0,Y 576.228,Z 702.013,A -85,B 0,C 180,E1 -9813.484,E2 -9813.484} C_VEL
LIN {X 0,Y 576.265,Z 697.714,A -85,B 0,C 180,E1 -9814.881,E2 -9814.881} C_VEL
LIN {X 0,Y 576.369,Z 693.427,A -85,B 0,C 180,E1 -9815.929,E2 -9815.929} C_VEL
LIN {X 0,Y 576.492,Z 687.112,A -85,B 0,C 180,E1 -9817.154,E2 -9817.154} C_VEL
LIN {X 0,Y 576.728,Z 679.197,A -85,B 0,C 180,E1 -9818.38,E2 -9818.38} C_VEL
LIN {X 0,Y 577.097,Z 670.907,A -85,B 0,C 180,E1 -9819.431,E2 -9819.431} C_VEL
LIN {X 0,Y 577.434,Z 660.904,A -85,B 0,C 180,E1 -9820.484,E2 -9820.484} C_VEL
LIN {X 0,Y 577.894,Z 649.761,A -85,B 0,C 180,E1 -9821.448,E2 -9821.448} C_VEL
LIN {X 0,Y 578.294,Z 638.673,A -85,B 0,C 180,E1 -9822.237,E2 -9822.237} C_VEL
LIN {X 0,Y 578.778,Z 626.63,A -85,B 0,C 180,E1 -9822.938,E2 -9822.938} C_VEL
LIN {X 0,Y 579.229,Z 613.385,A -85,B 0,C 180,E1 -9823.55,E2 -9823.55} C_VEL
LIN {X 0,Y 579.632,Z 599.788,A -85,B 0,C 180,E1 -9824.031,E2 -9824.031} C_VEL
LIN {X 0,Y 579.901,Z 587.053,A -85,B 0,C 180,E1 -9824.359,E2 -9824.359} C_VEL
LIN {X 0,Y 580.4,Z 570.349,A -85,B 0,C 180,E1 -9824.706,E2 -9824.706} C_VEL
LIN {X 0,Y 580.769,Z 524.104,A -85,B 0,C 180,E1 -9825.317,E2 -9825.317} C_VEL
LIN {X 0,Y 581.74,Z 462.911,A -85,B 0,C 180,E1 -9826.268,E2 -9826.268} C_VEL
LIN {X 0,Y 579.433,Z 438.437,A -85,B 0,C 180,E1 -9826.763,E2 -9826.763} C_VEL
LIN {X 0,Y 578.176,Z 427.43,A -85,B 0,C 180,E1 -9827.066,E2 -9827.066} C_VEL
LIN {X 0,Y 578.032,Z 425.785,A -85,B 0,C 180,E1 -9827.12,E2 -9827.12} C_VEL
LIN {X 0,Y 578.861,Z 397.295,A -85,B 0,C 180,E1 -9830.173,E2 -9830.173} C_VEL
LIN {X 0,Y 579.73,Z 371.913,A -85,B 0,C 180,E1 -9832.91,E2 -9832.91} C_VEL
LIN {X 0,Y 580.704,Z 345.963,A -85,B 0,C 180,E1 -9835.736,E2 -9835.736} C_VEL
LIN {X 0,Y 580.364,Z 340.714,A -85,B 0,C 180,E1 -9836.33,E2 -9836.33} C_VEL
LIN {X 0,Y 577.342,Z 326.13,A -85,B 0,C 180,E1 -9838.097,E2 -9838.097} C_VEL
LIN {X 0,Y 577.305,Z 326.128,A -85,B 0,C 180,E1 -9840.636,E2 -9840.636} C_VEL
LIN {X 0,Y 577.307,Z 326.132,A -85,B 0,C 180,E1 -9843.157,E2 -9843.157} C_VEL
LIN {X 0,Y 577.327,Z 326.127,A -85,B 0,C 180,E1 -9845.622,E2 -9845.622} C_VEL
LIN {X 0,Y 577.283,Z 326.131,A -85,B 0,C 180,E1 -9848.229,E2 -9848.229} C_VEL
LIN {X 0,Y 577.305,Z 326.132,A -85,B 0,C 180,E1 -9850.934,E2 -9850.934} C_VEL
LIN {X 0,Y 577.331,Z 326.128,A -85,B 0,C 180,E1 -9853.753,E2 -9853.753} C_VEL
LIN {X 0,Y 577.332,Z 326.127,A -85,B 0,C 180,E1 -9856.247,E2 -9856.247} C_VEL
LIN {X 0,Y 577.307,Z 326.132,A -85,B 0,C 180,E1 -9859.067,E2 -9859.067} C_VEL
LIN {X 0,Y 577.295,Z 326.129,A -85,B 0,C 180,E1 -9861.772,E2 -9861.772} C_VEL
LIN {X 0,Y 577.376,Z 326.125,A -85,B 0,C 180,E1 -9864.387,E2 -9864.387} C_VEL
LIN {X 0,Y 577.326,Z 326.133,A -85,B 0,C 180,E1 -9866.909,E2 -9866.909} C_VEL
LIN {X 0,Y 577.319,Z 326.139,A -85,B 0,C 180,E1 -9869.477,E2 -9869.477} C_VEL
LIN {X 0,Y 577.35,Z 326.144,A -85,B 0,C 180,E1 -9871.168,E2 -9871.168} C_VEL
LIN {X 0,Y 581.2,Z 340.35,A -85,B 0,C 180,E1 -9872.888,E2 -9872.888} C_VEL
LIN {X 0,Y 582.672,Z 348.146,A -85,B 0,C 180,E1 -9873.783,E2 -9873.783} C_VEL
LIN {X 0,Y 581.855,Z 372.945,A -85,B 0,C 180,E1 -9876.333,E2 -9876.333} C_VEL
LIN {X 0,Y 580.887,Z 400.6,A -85,B 0,C 180,E1 -9879.163,E2 -9879.163} C_VEL
LIN {X 0,Y 580.138,Z 425.414,A -85,B 0,C 180,E1 -9881.705,E2 -9881.705} C_VEL
LIN {X 0,Y 579.724,Z 439.601,A -85,B 0,C 180,E1 -9883.166,E2 -9883.166} C_VEL
LIN {X 0,Y 582.26,Z 457.184,A -85,B 0,C 180,E1 -9883.556,E2 -9883.556} C_VEL
LIN {X 0,Y 582.132,Z 473.821,A -85,B 0,C 180,E1 -9883.822,E2 -9883.822} C_VEL
LIN {X 0,Y 580.677,Z 569.985,A -85,B 0,C 180,E1 -9885.257,E2 -9885.257} C_VEL
LIN {X 0,Y 580.316,Z 585.681,A -85,B 0,C 180,E1 -9885.54,E2 -9885.54} C_VEL
LIN {X 0,Y 579.962,Z 599.676,A -85,B 0,C 180,E1 -9885.933,E2 -9885.933} C_VEL
LIN {X 0,Y 579.54,Z 613.364,A -85,B 0,C 180,E1 -9886.457,E2 -9886.457} C_VEL
LIN {X 0,Y 578.999,Z 627.305,A -85,B 0,C 180,E1 -9887.156,E2 -9887.156} C_VEL
LIN {X 0,Y 578.392,Z 639.821,A -85,B 0,C 180,E1 -9887.942,E2 -9887.942} C_VEL
LIN {X 0,Y 577.956,Z 651.198,A -85,B 0,C 180,E1 -9888.819,E2 -9888.819} C_VEL
LIN {X 0,Y 577.571,Z 660.675,A -85,B 0,C 180,E1 -9889.696,E2 -9889.696} C_VEL
LIN {X 0,Y 577.138,Z 670.198,A -85,B 0,C 180,E1 -9890.746,E2 -9890.746} C_VEL
LIN {X 0,Y 576.78,Z 679.307,A -85,B 0,C 180,E1 -9891.972,E2 -9891.972} C_VEL
LIN {X 0,Y 576.546,Z 685.685,A -85,B 0,C 180,E1 -9893.022,E2 -9893.022} C_VEL
LIN {X 0,Y 576.372,Z 690.917,A -85,B 0,C 180,E1 -9894.071,E2 -9894.071} C_VEL
LIN {X 0,Y 576.199,Z 696.279,A -85,B 0,C 180,E1 -9895.428,E2 -9895.428} C_VEL
LIN {X 0,Y 576.175,Z 699.436,A -85,B 0,C 180,E1 -9896.515,E2 -9896.515} C_VEL
LIN {X 0,Y 576.079,Z 702.217,A -85,B 0,C 180,E1 -9897.91,E2 -9897.91} C_VEL
LIN {X 0,Y 576.049,Z 703.577,A -85,B 0,C 180,E1 -9899.303,E2 -9899.303} C_VEL
LIN {X 0,Y 576.048,Z 703.515,A -85,B 0,C 180,E1 -9900.697,E2 -9900.697} C_VEL
LIN {X 0,Y 576.077,Z 702.053,A -85,B 0,C 180,E1 -9902.091,E2 -9902.091} C_VEL
LIN {X 0,Y 576.17,Z 699.174,A -85,B 0,C 180,E1 -9903.485,E2 -9903.485} C_VEL
LIN {X 0,Y 576.226,Z 694.804,A -85,B 0,C 180,E1 -9904.881,E2 -9904.881} C_VEL
LIN {X 0,Y 576.34,Z 690.443,A -85,B 0,C 180,E1 -9905.93,E2 -9905.93} C_VEL
LIN {X 0,Y 576.477,Z 684.071,A -85,B 0,C 180,E1 -9907.155,E2 -9907.155} C_VEL
LIN {X 0,Y 576.721,Z 676.127,A -85,B 0,C 180,E1 -9908.381,E2 -9908.381} C_VEL
LIN {X 0,Y 577.089,Z 667.809,A -85,B 0,C 180,E1 -9909.431,E2 -9909.431} C_VEL
LIN {X 0,Y 577.48,Z 657.787,A -85,B 0,C 180,E1 -9910.483,E2 -9910.483} C_VEL
LIN {X 0,Y 577.86,Z 646.57,A -85,B 0,C 180,E1 -9911.449,E2 -9911.449} C_VEL
LIN {X 0,Y 578.319,Z 634.089,A -85,B 0,C 180,E1 -9912.326,E2 -9912.326} C_VEL
LIN {X 0,Y 578.849,Z 621.794,A -85,B 0,C 180,E1 -9913.025,E2 -9913.025} C_VEL
LIN {X 0,Y 579.285,Z 608.24,A -85,B 0,C 180,E1 -9913.638,E2 -9913.638} C_VEL
LIN {X 0,Y 579.655,Z 594.084,A -85,B 0,C 180,E1 -9914.12,E2 -9914.12} C_VEL
LIN {X 0,Y 579.943,Z 580.299,A -85,B 0,C 180,E1 -9914.447,E2 -9914.447} C_VEL
LIN {X 0,Y 580.633,Z 520.899,A -85,B 0,C 180,E1 -9915.29,E2 -9915.29} C_VEL
LIN {X 0,Y 581.28,Z 456.949,A -85,B 0,C 180,E1 -9916.203,E2 -9916.203} C_VEL
LIN {X 0,Y 579.08,Z 439.622,A -85,B 0,C 180,E1 -9916.514,E2 -9916.514} C_VEL
LIN {X 0,Y 580.016,Z 408.249,A -85,B 0,C 180,E1 -9919.764,E2 -9919.764} C_VEL
LIN {X 0,Y 580.944,Z 378.266,A -85,B 0,C 180,E1 -9922.883,E2 -9922.883} C_VEL
LIN {X 0,Y 581.718,Z 353.796,A -85,B 0,C 180,E1 -9925.435,E2 -9925.435} C_VEL
LIN {X 0,Y 581.831,Z 345.992,A -85,B 0,C 180,E1 -9926.259,E2 -9926.259} C_VEL
LIN {X 0,Y 577.412,Z 326.119,A -85,B 0,C 180,E1 -9928.557,E2 -9928.557} C_VEL
LIN {X 0,Y 577.352,Z 326.129,A -85,B 0,C 180,E1 -9931.445,E2 -9931.445} C_VEL
LIN {X 0,Y 577.346,Z 326.122,A -85,B 0,C 180,E1 -9933.923,E2 -9933.923} C_VEL
LIN {X 0,Y 577.387,Z 326.116,A -85,B 0,C 180,E1 -9936.473,E2 -9936.473} C_VEL
LIN {X 0,Y 577.318,Z 326.134,A -85,B 0,C 180,E1 -9939.117,E2 -9939.117} C_VEL
LIN {X 0,Y 577.355,Z 326.12,A -85,B 0,C 180,E1 -9941.856,E2 -9941.856} C_VEL
LIN {X 0,Y 577.362,Z 326.125,A -85,B 0,C 180,E1 -9944.721,E2 -9944.721} C_VEL
LIN {X 0,Y 577.363,Z 326.119,A -85,B 0,C 180,E1 -9947.735,E2 -9947.735} C_VEL
LIN {X 0,Y 577.34,Z 326.123,A -85,B 0,C 180,E1 -9949.983,E2 -9949.983} C_VEL
LIN {X 0,Y 577.387,Z 326.118,A -85,B 0,C 180,E1 -9953.194,E2 -9953.194} C_VEL
LIN {X 0,Y 577.366,Z 326.119,A -85,B 0,C 180,E1 -9955.585,E2 -9955.585} C_VEL
LIN {X 0,Y 577.343,Z 326.126,A -85,B 0,C 180,E1 -9958.255,E2 -9958.255} C_VEL
LIN {X 0,Y 576.67,Z 326.213,A -85,B 0,C 180,E1 -9958.836,E2 -9958.836} C_VEL
LIN {X 0,Y 573.805,Z 326.568,A -85,B 0,C 180,E1 -9959.78,E2 -9959.78} C_VEL
LIN {X 0,Y 571.401,Z 326.869,A -85,B 0,C 180,E1 -9960.54,E2 -9960.54} C_VEL
LIN {X 0,Y 570.391,Z 326.989,A -85,B 0,C 180,E1 -9961.127,E2 -9961.127} C_VEL
LIN {X 0,Y 570.321,Z 326.997,A -85,B 0,C 180,E1 -9961.325,E2 -9961.325} C_VEL
LIN {X 0,Y 570.282,Z 327.003,A -85,B 0,C 180,E1 -9963.758,E2 -9963.758} C_VEL
LIN {X 0,Y 570.323,Z 327.003,A -85,B 0,C 180,E1 -9966.091,E2 -9966.091} C_VEL
LIN {X 0,Y 570.362,Z 326.992,A -85,B 0,C 180,E1 -9969.137,E2 -9969.137} C_VEL
LIN {X 0,Y 570.336,Z 327.002,A -85,B 0,C 180,E1 -9972.12,E2 -9972.12} C_VEL
LIN {X 0,Y 570.332,Z 326.998,A -85,B 0,C 180,E1 -9975.054,E2 -9975.054} C_VEL
LIN {X 0,Y 570.341,Z 326.997,A -85,B 0,C 180,E1 -9977.229,E2 -9977.229} C_VEL
LIN {X 0,Y 570.379,Z 326.992,A -85,B 0,C 180,E1 -9978.588,E2 -9978.588} C_VEL
LIN {X 0,Y 574.785,Z 340.602,A -85,B 0,C 180,E1 -9978.884,E2 -9978.884} C_VEL
LIN {X 0,Y 574.138,Z 445.913,A -85,B 0,C 180,E1 -9980.21,E2 -9980.21} C_VEL
LIN {X 0,Y 574.034,Z 460.083,A -85,B 0,C 180,E1 -9980.496,E2 -9980.496} C_VEL
LIN {X 0,Y 573.846,Z 473.766,A -85,B 0,C 180,E1 -9980.914,E2 -9980.914} C_VEL
LIN {X 0,Y 573.491,Z 487.508,A -85,B 0,C 180,E1 -9981.484,E2 -9981.484} C_VEL
LIN {X 0,Y 573.125,Z 500.376,A -85,B 0,C 180,E1 -9982.18,E2 -9982.18} C_VEL
LIN {X 0,Y 572.7,Z 512.173,A -85,B 0,C 180,E1 -9982.975,E2 -9982.975} C_VEL
LIN {X 0,Y 572.142,Z 522.889,A -85,B 0,C 180,E1 -9983.851,E2 -9983.851} C_VEL
LIN {X 0,Y 571.589,Z 533.462,A -85,B 0,C 180,E1 -9984.903,E2 -9984.903} C_VEL
LIN {X 0,Y 571.176,Z 542.188,A -85,B 0,C 180,E1 -9985.957,E2 -9985.957} C_VEL
LIN {X 0,Y 570.776,Z 550.549,A -85,B 0,C 180,E1 -9987.186,E2 -9987.186} C_VEL
LIN {X 0,Y 570.474,Z 556.418,A -85,B 0,C 180,E1 -9988.241,E2 -9988.241} C_VEL
LIN {X 0,Y 570.118,Z 562.684,A -85,B 0,C 180,E1 -9989.648,E2 -9989.648} C_VEL
LIN {X 0,Y 569.876,Z 566.323,A -85,B 0,C 180,E1 -9990.704,E2 -9990.704} C_VEL
LIN {X 0,Y 569.832,Z 569.871,A -85,B 0,C 180,E1 -9992.113,E2 -9992.113} C_VEL
LIN {X 0,Y 569.859,Z 572.065,A -85,B 0,C 180,E1 -9993.524,E2 -9993.524} C_VEL
LIN {X 0,Y 569.741,Z 572.982,A -85,B 0,C 180,E1 -9994.937,E2 -9994.937} C_VEL
LIN {X 0,Y 569.849,Z 572.59,A -85,B 0,C 180,E1 -9996.352,E2 -9996.352} C_VEL
LIN {X 0,Y 569.928,Z 570.906,A -85,B 0,C 180,E1 -9997.77,E2 -9997.77} C_VEL
LIN {X 0,Y 570.075,Z 567.874,A -85,B 0,C 180,E1 -9999.191,E2 -9999.191} C_VEL
LIN {X 0,Y 570.374,Z 564.601,A -85,B 0,C 180,E1 -10000.257,E2 -10000.257} C_VEL
LIN {X 0,Y 570.695,Z 558.913,A -85,B 0,C 180,E1 -10001.684,E2 -10001.684} C_VEL
LIN {X 0,Y 571.136,Z 552.468,A -85,B 0,C 180,E1 -10002.934,E2 -10002.934} C_VEL
LIN {X 0,Y 571.64,Z 544.434,A -85,B 0,C 180,E1 -10004.186,E2 -10004.186} C_VEL
LIN {X 0,Y 572.159,Z 535.988,A -85,B 0,C 180,E1 -10005.261,E2 -10005.261} C_VEL
LIN {X 0,Y 572.717,Z 525.708,A -85,B 0,C 180,E1 -10006.338,E2 -10006.338} C_VEL
LIN {X 0,Y 573.256,Z 515.972,A -85,B 0,C 180,E1 -10007.185,E2 -10007.185} C_VEL
LIN {X 0,Y 573.708,Z 505.415,A -85,B 0,C 180,E1 -10007.956,E2 -10007.956} C_VEL
LIN {X 0,Y 574.237,Z 493.293,A -85,B 0,C 180,E1 -10008.675,E2 -10008.675} C_VEL
LIN {X 0,Y 574.56,Z 480.898,A -85,B 0,C 180,E1 -10009.264,E2 -10009.264} C_VEL
LIN {X 0,Y 574.842,Z 467.806,A -85,B 0,C 180,E1 -10009.74,E2 -10009.74} C_VEL
LIN {X 0,Y 575.013,Z 453.502,A -85,B 0,C 180,E1 -10010.108,E2 -10010.108} C_VEL
LIN {X 0,Y 575.127,Z 434.707,A -85,B 0,C 180,E1 -10010.392,E2 -10010.392} C_VEL
LIN {X 0,Y 575.797,Z 341.629,A -85,B 0,C 180,E1 -10011.569,E2 -10011.569} C_VEL
LIN {X 0,Y 570.294,Z 327.011,A -85,B 0,C 180,E1 -10011.954,E2 -10011.954} C_VEL
LIN {X 0,Y 570.324,Z 327.009,A -85,B 0,C 180,E1 -10014.682,E2 -10014.682} C_VEL
LIN {X 0,Y 570.294,Z 327.006,A -85,B 0,C 180,E1 -10017.832,E2 -10017.832} C_VEL
LIN {X 0,Y 570.277,Z 327.006,A -85,B 0,C 180,E1 -10020.708,E2 -10020.708} C_VEL
LIN {X 0,Y 570.267,Z 327.004,A -85,B 0,C 180,E1 -10023.36,E2 -10023.36} C_VEL
LIN {X 0,Y 570.285,Z 327.008,A -85,B 0,C 180,E1 -10026.126,E2 -10026.126} C_VEL
LIN {X 0,Y 570.26,Z 327.005,A -85,B 0,C 180,E1 -10029.301,E2 -10029.301} C_VEL
LIN {X 0,Y 570.268,Z 327.007,A -85,B 0,C 180,E1 -10031.55,E2 -10031.55} C_VEL
LIN {X 0,Y 570.314,Z 326.999,A -85,B 0,C 180,E1 -10034.574,E2 -10034.574} C_VEL
LIN {X 0,Y 570.313,Z 327,A -85,B 0,C 180,E1 -10037.507,E2 -10037.507} C_VEL
LIN {X 0,Y 570.281,Z 327.003,A -85,B 0,C 180,E1 -10040.306,E2 -10040.306} C_VEL
LIN {X 0,Y 570.27,Z 326.985,A -85,B 0,C 180,E1 -10042.997,E2 -10042.997} C_VEL
LIN {X 0,Y 570.283,Z 326.997,A -85,B 0,C 180,E1 -10045.598,E2 -10045.598} C_VEL
LIN {X 0,Y 570.311,Z 326.999,A -85,B 0,C 180,E1 -10048.121,E2 -10048.121} C_VEL
LIN {X 0,Y 570.291,Z 327.002,A -85,B 0,C 180,E1 -10051.379,E2 -10051.379} C_VEL
LIN {X 0,Y 570.283,Z 327.003,A -85,B 0,C 180,E1 -10053.758,E2 -10053.758} C_VEL
LIN {X 0,Y 570.295,Z 327.004,A -85,B 0,C 180,E1 -10056.089,E2 -10056.089} C_VEL
LIN {X 0,Y 570.319,Z 326.994,A -85,B 0,C 180,E1 -10059.135,E2 -10059.135} C_VEL
LIN {X 0,Y 570.31,Z 327.008,A -85,B 0,C 180,E1 -10062.118,E2 -10062.118} C_VEL
LIN {X 0,Y 570.307,Z 327.006,A -85,B 0,C 180,E1 -10062.748,E2 -10062.748} C_VEL
LIN {X 0,Y 574.255,Z 340.124,A -85,B 0,C 180,E1 -10063.053,E2 -10063.053} C_VEL
LIN {X 0,Y 573.147,Z 447.589,A -85,B 0,C 180,E1 -10064.6,E2 -10064.6} C_VEL
LIN {X 0,Y 572.974,Z 462.736,A -85,B 0,C 180,E1 -10064.971,E2 -10064.971} C_VEL
LIN {X 0,Y 572.751,Z 477.237,A -85,B 0,C 180,E1 -10065.481,E2 -10065.481} C_VEL
LIN {X 0,Y 572.423,Z 490.645,A -85,B 0,C 180,E1 -10066.105,E2 -10066.105} C_VEL
LIN {X 0,Y 572.09,Z 502.813,A -85,B 0,C 180,E1 -10066.818,E2 -10066.818} C_VEL
LIN {X 0,Y 571.646,Z 515.155,A -85,B 0,C 180,E1 -10067.708,E2 -10067.708} C_VEL
LIN {X 0,Y 571.232,Z 526.282,A -85,B 0,C 180,E1 -10068.685,E2 -10068.685} C_VEL
LIN {X 0,Y 570.967,Z 536.246,A -85,B 0,C 180,E1 -10069.753,E2 -10069.753} C_VEL
LIN {X 0,Y 570.572,Z 544.496,A -85,B 0,C 180,E1 -10070.817,E2 -10070.817} C_VEL
LIN {X 0,Y 570.288,Z 552.369,A -85,B 0,C 180,E1 -10072.057,E2 -10072.057} C_VEL
LIN {X 0,Y 570.045,Z 558.688,A -85,B 0,C 180,E1 -10073.296,E2 -10073.296} C_VEL
LIN {X 0,Y 569.84,Z 564.086,A -85,B 0,C 180,E1 -10074.656,E2 -10074.656} C_VEL
LIN {X 0,Y 569.767,Z 567.374,A -85,B 0,C 180,E1 -10075.77,E2 -10075.77} C_VEL
LIN {X 0,Y 569.787,Z 570.255,A -85,B 0,C 180,E1 -10077.181,E2 -10077.181} C_VEL
LIN {X 0,Y 569.653,Z 571.741,A -85,B 0,C 180,E1 -10078.591,E2 -10078.591} C_VEL
LIN {X 0,Y 569.573,Z 571.826,A -85,B 0,C 180,E1 -10080,E2 -10080} C_VEL
LIN {X 0,Y 569.679,Z 570.522,A -85,B 0,C 180,E1 -10081.409,E2 -10081.409} C_VEL
LIN {X 0,Y 570.017,Z 567.802,A -85,B 0,C 180,E1 -10082.817,E2 -10082.817} C_VEL
LIN {X 0,Y 570.426,Z 563.609,A -85,B 0,C 180,E1 -10084.225,E2 -10084.225} C_VEL
LIN {X 0,Y 570.394,Z 559.424,A -85,B 0,C 180,E1 -10085.284,E2 -10085.284} C_VEL
LIN {X 0,Y 570.806,Z 554.197,A -85,B 0,C 180,E1 -10086.341,E2 -10086.341} C_VEL
LIN {X 0,Y 571.256,Z 546.704,A -85,B 0,C 180,E1 -10087.574,E2 -10087.574} C_VEL
LIN {X 0,Y 571.587,Z 538.839,A -85,B 0,C 180,E1 -10088.634,E2 -10088.634} C_VEL
LIN {X 0,Y 572.009,Z 529.319,A -85,B 0,C 180,E1 -10089.693,E2 -10089.693} C_VEL
LIN {X 0,Y 572.369,Z 518.707,A -85,B 0,C 180,E1 -10090.666,E2 -10090.666} C_VEL
LIN {X 0,Y 572.93,Z 508.196,A -85,B 0,C 180,E1 -10091.459,E2 -10091.459} C_VEL
LIN {X 0,Y 573.482,Z 496.25,A -85,B 0,C 180,E1 -10092.199,E2 -10092.199} C_VEL
LIN {X 0,Y 573.804,Z 482.748,A -85,B 0,C 180,E1 -10092.872,E2 -10092.872} C_VEL
LIN {X 0,Y 574.079,Z 468.613,A -85,B 0,C 180,E1 -10093.404,E2 -10093.404} C_VEL
LIN {X 0,Y 574.22,Z 454.512,A -85,B 0,C 180,E1 -10093.783,E2 -10093.783} C_VEL
LIN {X 0,Y 574.441,Z 430.247,A -85,B 0,C 180,E1 -10094.182,E2 -10094.182} C_VEL
LIN {X 0,Y 575.957,Z 341.206,A -85,B 0,C 180,E1 -10095.561,E2 -10095.561} C_VEL
LIN {X 0,Y 570.496,Z 327.747,A -85,B 0,C 180,E1 -10096.014,E2 -10096.014} C_VEL
LIN {X 0,Y 570.368,Z 327.001,A -85,B 0,C 180,E1 -10096.034,E2 -10096.034} C_VEL
LIN {X 0,Y 570.341,Z 326.999,A -85,B 0,C 180,E1 -10098.976,E2 -10098.976} C_VEL
LIN {X 0,Y 570.336,Z 327.002,A -85,B 0,C 180,E1 -10101.619,E2 -10101.619} C_VEL
LIN {X 0,Y 570.336,Z 327.004,A -85,B 0,C 180,E1 -10103.909,E2 -10103.909} C_VEL
LIN {X 0,Y 570.291,Z 327.004,A -85,B 0,C 180,E1 -10107.029,E2 -10107.029} C_VEL
LIN {X 0,Y 570.313,Z 327.003,A -85,B 0,C 180,E1 -10109.424,E2 -10109.424} C_VEL
LIN {X 0,Y 570.31,Z 327.002,A -85,B 0,C 180,E1 -10112.064,E2 -10112.064} C_VEL
LIN {X 0,Y 570.34,Z 326.994,A -85,B 0,C 180,E1 -10114.63,E2 -10114.63} C_VEL
LIN {X 0,Y 570.319,Z 326.998,A -85,B 0,C 180,E1 -10117.031,E2 -10117.031} C_VEL
LIN {X 0,Y 570.28,Z 327.002,A -85,B 0,C 180,E1 -10119.694,E2 -10119.694} C_VEL
LIN {X 0,Y 570.295,Z 326.997,A -85,B 0,C 180,E1 -10122.529,E2 -10122.529} C_VEL
LIN {X 0,Y 570.312,Z 326.999,A -85,B 0,C 180,E1 -10125.568,E2 -10125.568} C_VEL
LIN {X 0,Y 570.272,Z 327.005,A -85,B 0,C 180,E1 -10128.525,E2 -10128.525} C_VEL
LIN {X 0,Y 570.263,Z 327.008,A -85,B 0,C 180,E1 -10131.213,E2 -10131.213} C_VEL
LIN {X 0,Y 570.284,Z 327.005,A -85,B 0,C 180,E1 -10134.158,E2 -10134.158} C_VEL
LIN {X 0,Y 570.266,Z 327.008,A -85,B 0,C 180,E1 -10137.286,E2 -10137.286} C_VEL
LIN {X 0,Y 570.263,Z 327.006,A -85,B 0,C 180,E1 -10139.762,E2 -10139.762} C_VEL
LIN {X 0,Y 570.348,Z 327.137,A -85,B 0,C 180,E1 -10141.232,E2 -10141.232} C_VEL
LIN {X 0,Y 574.033,Z 343.92,A -85,B 0,C 180,E1 -10143.357,E2 -10143.357} C_VEL
LIN {X 0,Y 574.465,Z 347.332,A -85,B 0,C 180,E1 -10143.768,E2 -10143.768} C_VEL
LIN {X 0,Y 573.563,Z 367.485,A -85,B 0,C 180,E1 -10146.043,E2 -10146.043} C_VEL
LIN {X 0,Y 572.424,Z 394.271,A -85,B 0,C 180,E1 -10149.028,E2 -10149.028} C_VEL
LIN {X 0,Y 571.547,Z 415.954,A -85,B 0,C 180,E1 -10151.419,E2 -10151.419} C_VEL
LIN {X 0,Y 571.146,Z 430.317,A -85,B 0,C 180,E1 -10152.992,E2 -10152.992} C_VEL
LIN {X 0,Y 574.347,Z 457.423,A -85,B 0,C 180,E1 -10153.443,E2 -10153.443} C_VEL
LIN {X 0,Y 575.019,Z 465.976,A -85,B 0,C 180,E1 -10153.574,E2 -10153.574} C_VEL
LIN {X 0,Y 573.998,Z 569.967,A -85,B 0,C 180,E1 -10154.892,E2 -10154.892} C_VEL
LIN {X 0,Y 573.516,Z 584.12,A -85,B 0,C 180,E1 -10155.207,E2 -10155.207} C_VEL
LIN {X 0,Y 572.913,Z 598.185,A -85,B 0,C 180,E1 -10155.666,E2 -10155.666} C_VEL
LIN {X 0,Y 572.224,Z 612.156,A -85,B 0,C 180,E1 -10156.281,E2 -10156.281} C_VEL
LIN {X 0,Y 571.614,Z 624.688,A -85,B 0,C 180,E1 -10156.987,E2 -10156.987} C_VEL
LIN {X 0,Y 570.796,Z 644.113,A -85,B 0,C 180,E1 -10158.228,E2 -10158.228} C_VEL
LIN {X 0,Y 570.412,Z 655.596,A -85,B 0,C 180,E1 -10159.138,E2 -10159.138} C_VEL
LIN {X 0,Y 569.998,Z 665.583,A -85,B 0,C 180,E1 -10160.093,E2 -10160.093} C_VEL
LIN {X 0,Y 569.721,Z 674.816,A -85,B 0,C 180,E1 -10161.16,E2 -10161.16} C_VEL
LIN {X 0,Y 569.436,Z 683.607,A -85,B 0,C 180,E1 -10162.401,E2 -10162.401} C_VEL
LIN {X 0,Y 569.293,Z 690.667,A -85,B 0,C 180,E1 -10163.642,E2 -10163.642} C_VEL
LIN {X 0,Y 569.234,Z 695.505,A -85,B 0,C 180,E1 -10164.705,E2 -10164.705} C_VEL
LIN {X 0,Y 569.106,Z 700.471,A -85,B 0,C 180,E1 -10166.118,E2 -10166.118} C_VEL
LIN {X 0,Y 569.119,Z 703.125,A -85,B 0,C 180,E1 -10167.178,E2 -10167.178} C_VEL
LIN {X 0,Y 569.058,Z 705.393,A -85,B 0,C 180,E1 -10168.589,E2 -10168.589} C_VEL
LIN {X 0,Y 569.053,Z 706.236,A -85,B 0,C 180,E1 -10170,E2 -10170} C_VEL
LIN {X 0,Y 569.058,Z 705.657,A -85,B 0,C 180,E1 -10171.411,E2 -10171.411} C_VEL
LIN {X 0,Y 569.119,Z 703.624,A -85,B 0,C 180,E1 -10172.822,E2 -10172.822} C_VEL
LIN {X 0,Y 569.123,Z 700.107,A -85,B 0,C 180,E1 -10174.235,E2 -10174.235} C_VEL
LIN {X 0,Y 569.267,Z 695.014,A -85,B 0,C 180,E1 -10175.649,E2 -10175.649} C_VEL
LIN {X 0,Y 569.387,Z 690.066,A -85,B 0,C 180,E1 -10176.711,E2 -10176.711} C_VEL
LIN {X 0,Y 569.615,Z 682.899,A -85,B 0,C 180,E1 -10177.952,E2 -10177.952} C_VEL
LIN {X 0,Y 569.852,Z 675.367,A -85,B 0,C 180,E1 -10179.016,E2 -10179.016} C_VEL
LIN {X 0,Y 570.253,Z 666.282,A -85,B 0,C 180,E1 -10180.081,E2 -10180.081} C_VEL
LIN {X 0,Y 570.71,Z 655.374,A -85,B 0,C 180,E1 -10181.136,E2 -10181.136} C_VEL
LIN {X 0,Y 571.177,Z 644.084,A -85,B 0,C 180,E1 -10182.033,E2 -10182.033} C_VEL
LIN {X 0,Y 571.625,Z 631.728,A -85,B 0,C 180,E1 -10182.832,E2 -10182.832} C_VEL
LIN {X 0,Y 572.158,Z 619.867,A -85,B 0,C 180,E1 -10183.45,E2 -10183.45} C_VEL
LIN {X 0,Y 572.581,Z 605.769,A -85,B 0,C 180,E1 -10184.026,E2 -10184.026} C_VEL
LIN {X 0,Y 572.937,Z 590.945,A -85,B 0,C 180,E1 -10184.469,E2 -10184.469} C_VEL
LIN {X 0,Y 573.289,Z 576.071,A -85,B 0,C 180,E1 -10184.754,E2 -10184.754} C_VEL
LIN {X 0,Y 573.533,Z 559.262,A -85,B 0,C 180,E1 -10185.012,E2 -10185.012} C_VEL
LIN {X 0,Y 574.935,Z 475.677,A -85,B 0,C 180,E1 -10186.305,E2 -10186.305} C_VEL
LIN {X 0,Y 574.969,Z 462.14,A -85,B 0,C 180,E1 -10186.533,E2 -10186.533} C_VEL
LIN {X 0,Y 572.714,Z 438.144,A -85,B 0,C 180,E1 -10187.037,E2 -10187.037} C_VEL
LIN {X 0,Y 571.145,Z 424.689,A -85,B 0,C 180,E1 -10187.435,E2 -10187.435} C_VEL
LIN {X 0,Y 571.088,Z 423.434,A -85,B 0,C 180,E1 -10187.487,E2 -10187.487} C_VEL
LIN {X 0,Y 571.924,Z 396.323,A -85,B 0,C 180,E1 -10190.429,E2 -10190.429} C_VEL
LIN {X 0,Y 572.75,Z 372.432,A -85,B 0,C 180,E1 -10193.038,E2 -10193.038} C_VEL
LIN {X 0,Y 573.796,Z 346.695,A -85,B 0,C 180,E1 -10195.875,E2 -10195.875} C_VEL
LIN {X 0,Y 573.302,Z 341.595,A -85,B 0,C 180,E1 -10196.465,E2 -10196.465} C_VEL
LIN {X 0,Y 570.322,Z 327.004,A -85,B 0,C 180,E1 -10198.251,E2 -10198.251} C_VEL
LIN {X 0,Y 570.274,Z 327.005,A -85,B 0,C 180,E1 -10201.056,E2 -10201.056} C_VEL
LIN {X 0,Y 570.256,Z 327.01,A -85,B 0,C 180,E1 -10203.555,E2 -10203.555} C_VEL
LIN {X 0,Y 570.265,Z 327.006,A -85,B 0,C 180,E1 -10206.127,E2 -10206.127} C_VEL
LIN {X 0,Y 570.252,Z 327.008,A -85,B 0,C 180,E1 -10209.301,E2 -10209.301} C_VEL
LIN {X 0,Y 570.263,Z 327.008,A -85,B 0,C 180,E1 -10211.55,E2 -10211.55} C_VEL
LIN {X 0,Y 570.31,Z 327.004,A -85,B 0,C 180,E1 -10214.574,E2 -10214.574} C_VEL
LIN {X 0,Y 570.257,Z 327.011,A -85,B 0,C 180,E1 -10217.502,E2 -10217.502} C_VEL
LIN {X 0,Y 570.277,Z 327.006,A -85,B 0,C 180,E1 -10220.306,E2 -10220.306} C_VEL
LIN {X 0,Y 570.305,Z 327.005,A -85,B 0,C 180,E1 -10223,E2 -10223} C_VEL
LIN {X 0,Y 570.306,Z 327.003,A -85,B 0,C 180,E1 -10225.6,E2 -10225.6} C_VEL
LIN {X 0,Y 570.315,Z 327.008,A -85,B 0,C 180,E1 -10228.122,E2 -10228.122} C_VEL
LIN {X 0,Y 570.312,Z 327.11,A -85,B 0,C 180,E1 -10230.82,E2 -10230.82} C_VEL
LIN {X 0,Y 574.22,Z 340.918,A -85,B 0,C 180,E1 -10232.54,E2 -10232.54} C_VEL
LIN {X 0,Y 576.037,Z 350.383,A -85,B 0,C 180,E1 -10233.652,E2 -10233.652} C_VEL
LIN {X 0,Y 575.145,Z 375.946,A -85,B 0,C 180,E1 -10236.304,E2 -10236.304} C_VEL
LIN {X 0,Y 574.101,Z 402.919,A -85,B 0,C 180,E1 -10239.092,E2 -10239.092} C_VEL
LIN {X 0,Y 573.258,Z 429.453,A -85,B 0,C 180,E1 -10241.846,E2 -10241.846} C_VEL
LIN {X 0,Y 572.926,Z 439.584,A -85,B 0,C 180,E1 -10242.895,E2 -10242.895} C_VEL
LIN {X 0,Y 575.316,Z 455.824,A -85,B 0,C 180,E1 -10243.273,E2 -10243.273} C_VEL
LIN {X 0,Y 575.746,Z 461.658,A -85,B 0,C 180,E1 -10243.388,E2 -10243.388} C_VEL
LIN {X 0,Y 574.083,Z 554.62,A -85,B 0,C 180,E1 -10244.823,E2 -10244.823} C_VEL
LIN {X 0,Y 573.641,Z 581.818,A -85,B 0,C 180,E1 -10245.255,E2 -10245.255} C_VEL
LIN {X 0,Y 573.234,Z 596.194,A -85,B 0,C 180,E1 -10245.629,E2 -10245.629} C_VEL
LIN {X 0,Y 572.779,Z 609.637,A -85,B 0,C 180,E1 -10246.114,E2 -10246.114} C_VEL
LIN {X 0,Y 572.284,Z 622.818,A -85,B 0,C 180,E1 -10246.733,E2 -10246.733} C_VEL
LIN {X 0,Y 571.717,Z 634.872,A -85,B 0,C 180,E1 -10247.44,E2 -10247.44} C_VEL
LIN {X 0,Y 571.156,Z 647.161,A -85,B 0,C 180,E1 -10248.326,E2 -10248.326} C_VEL
LIN {X 0,Y 570.691,Z 657.486,A -85,B 0,C 180,E1 -10249.231,E2 -10249.231} C_VEL
LIN {X 0,Y 570.262,Z 667.402,A -85,B 0,C 180,E1 -10250.277,E2 -10250.277} C_VEL
LIN {X 0,Y 569.855,Z 675.785,A -85,B 0,C 180,E1 -10251.34,E2 -10251.34} C_VEL
LIN {X 0,Y 569.534,Z 683.784,A -85,B 0,C 180,E1 -10252.581,E2 -10252.581} C_VEL
LIN {X 0,Y 569.354,Z 689.396,A -85,B 0,C 180,E1 -10253.643,E2 -10253.643} C_VEL
LIN {X 0,Y 569.143,Z 695.255,A -85,B 0,C 180,E1 -10255.058,E2 -10255.058} C_VEL
LIN {X 0,Y 569.093,Z 699.511,A -85,B 0,C 180,E1 -10256.472,E2 -10256.472} C_VEL
LIN {X 0,Y 568.998,Z 702.276,A -85,B 0,C 180,E1 -10257.884,E2 -10257.884} C_VEL
LIN {X 0,Y 568.955,Z 703.605,A -85,B 0,C 180,E1 -10259.295,E2 -10259.295} C_VEL
LIN {X 0,Y 568.954,Z 703.51,A -85,B 0,C 180,E1 -10260.706,E2 -10260.706} C_VEL
LIN {X 0,Y 568.996,Z 702.016,A -85,B 0,C 180,E1 -10262.117,E2 -10262.117} C_VEL
LIN {X 0,Y 569.07,Z 699.1,A -85,B 0,C 180,E1 -10263.529,E2 -10263.529} C_VEL
LIN {X 0,Y 569.15,Z 694.688,A -85,B 0,C 180,E1 -10264.942,E2 -10264.942} C_VEL
LIN {X 0,Y 569.242,Z 690.278,A -85,B 0,C 180,E1 -10266.004,E2 -10266.004} C_VEL
LIN {X 0,Y 569.422,Z 683.853,A -85,B 0,C 180,E1 -10267.244,E2 -10267.244} C_VEL
LIN {X 0,Y 569.664,Z 675.844,A -85,B 0,C 180,E1 -10268.485,E2 -10268.485} C_VEL
LIN {X 0,Y 570.064,Z 667.455,A -85,B 0,C 180,E1 -10269.548,E2 -10269.548} C_VEL
LIN {X 0,Y 570.453,Z 657.316,A -85,B 0,C 180,E1 -10270.614,E2 -10270.614} C_VEL
LIN {X 0,Y 570.844,Z 645.976,A -85,B 0,C 180,E1 -10271.591,E2 -10271.591} C_VEL
LIN {X 0,Y 571.339,Z 633.362,A -85,B 0,C 180,E1 -10272.479,E2 -10272.479} C_VEL
LIN {X 0,Y 571.868,Z 620.898,A -85,B 0,C 180,E1 -10273.187,E2 -10273.187} C_VEL
LIN {X 0,Y 572.379,Z 607.084,A -85,B 0,C 180,E1 -10273.806,E2 -10273.806} C_VEL
LIN {X 0,Y 572.681,Z 593.19,A -85,B 0,C 180,E1 -10274.273,E2 -10274.273} C_VEL
LIN {X 0,Y 573.002,Z 579.025,A -85,B 0,C 180,E1 -10274.603,E2 -10274.603} C_VEL
LIN {X 0,Y 574.364,Z 457.516,A -85,B 0,C 180,E1 -10276.364,E2 -10276.364} C_VEL
LIN {X 0,Y 572.145,Z 439.555,A -85,B 0,C 180,E1 -10276.697,E2 -10276.697} C_VEL
LIN {X 0,Y 573.1,Z 407.777,A -85,B 0,C 180,E1 -10280.012,E2 -10280.012} C_VEL
LIN {X 0,Y 574.017,Z 379.418,A -85,B 0,C 180,E1 -10282.985,E2 -10282.985} C_VEL
LIN {X 0,Y 574.864,Z 354.352,A -85,B 0,C 180,E1 -10285.623,E2 -10285.623} C_VEL
LIN {X 0,Y 575.019,Z 348.85,A -85,B 0,C 180,E1 -10286.204,E2 -10286.204} C_VEL
LIN {X 0,Y 573.118,Z 339.42,A -85,B 0,C 180,E1 -10287.278,E2 -10287.278} C_VEL
LIN {X 0,Y 570.373,Z 326.996,A -85,B 0,C 180,E1 -10288.717,E2 -10288.717} C_VEL
LIN {X 0,Y 570.327,Z 326.997,A -85,B 0,C 180,E1 -10291.878,E2 -10291.878} C_VEL
LIN {X 0,Y 570.341,Z 326.995,A -85,B 0,C 180,E1 -10294.63,E2 -10294.63} C_VEL
LIN {X 0,Y 570.32,Z 327.003,A -85,B 0,C 180,E1 -10297.031,E2 -10297.031} C_VEL
LIN {X 0,Y 570.289,Z 327.002,A -85,B 0,C 180,E1 -10299.694,E2 -10299.694} C_VEL
LIN {X 0,Y 570.329,Z 326.998,A -85,B 0,C 180,E1 -10302.533,E2 -10302.533} C_VEL
LIN {X 0,Y 570.315,Z 326.998,A -85,B 0,C 180,E1 -10305.568,E2 -10305.568} C_VEL
LIN {X 0,Y 570.307,Z 327.003,A -85,B 0,C 180,E1 -10308.521,E2 -10308.521} C_VEL
LIN {X 0,Y 570.272,Z 327.005,A -85,B 0,C 180,E1 -10311.214,E2 -10311.214} C_VEL
LIN {X 0,Y 570.37,Z 326.993,A -85,B 0,C 180,E1 -10314.147,E2 -10314.147} C_VEL
LIN {X 0,Y 570.315,Z 327.005,A -85,B 0,C 180,E1 -10316.633,E2 -10316.633} C_VEL
LIN {X 0,Y 570.298,Z 327,A -85,B 0,C 180,E1 -10319.289,E2 -10319.289} C_VEL
LIN {X 0,Y 570.321,Z 326.997,A -85,B 0,C 180,E1 -10321.325,E2 -10321.325} C_VEL
LIN {X 0,Y 569.675,Z 327.081,A -85,B 0,C 180,E1 -10321.915,E2 -10321.915} C_VEL
LIN {X 0,Y 566.786,Z 327.444,A -85,B 0,C 180,E1 -10322.871,E2 -10322.871} C_VEL
LIN {X 0,Y 564.337,Z 327.751,A -85,B 0,C 180,E1 -10323.64,E2 -10323.64} C_VEL
LIN {X 0,Y 563.298,Z 327.879,A -85,B 0,C 180,E1 -10324.235,E2 -10324.235} C_VEL
LIN {X 0,Y 563.222,Z 327.885,A -85,B 0,C 180,E1 -10324.436,E2 -10324.436} C_VEL
LIN {X 0,Y 563.296,Z 327.872,A -85,B 0,C 180,E1 -10327.327,E2 -10327.327} C_VEL
LIN {X 0,Y 563.281,Z 327.876,A -85,B 0,C 180,E1 -10329.624,E2 -10329.624} C_VEL
LIN {X 0,Y 563.305,Z 327.877,A -85,B 0,C 180,E1 -10331.889,E2 -10331.889} C_VEL
LIN {X 0,Y 563.306,Z 327.871,A -85,B 0,C 180,E1 -10334.863,E2 -10334.863} C_VEL
LIN {X 0,Y 563.297,Z 327.873,A -85,B 0,C 180,E1 -10337.066,E2 -10337.066} C_VEL
LIN {X 0,Y 563.345,Z 327.87,A -85,B 0,C 180,E1 -10338.396,E2 -10338.396} C_VEL
LIN {X 0,Y 567.805,Z 341.114,A -85,B 0,C 180,E1 -10338.698,E2 -10338.698} C_VEL
LIN {X 0,Y 567.694,Z 379.73,A -85,B 0,C 180,E1 -10339.191,E2 -10339.191} C_VEL
LIN {X 0,Y 567.272,Z 446.586,A -85,B 0,C 180,E1 -10340.046,E2 -10340.046} C_VEL
LIN {X 0,Y 567.16,Z 460.791,A -85,B 0,C 180,E1 -10340.335,E2 -10340.335} C_VEL
LIN {X 0,Y 566.956,Z 474.492,A -85,B 0,C 180,E1 -10340.758,E2 -10340.758} C_VEL
LIN {X 0,Y 566.627,Z 487.277,A -85,B 0,C 180,E1 -10341.29,E2 -10341.29} C_VEL
LIN {X 0,Y 566.23,Z 500.23,A -85,B 0,C 180,E1 -10341.984,E2 -10341.984} C_VEL
LIN {X 0,Y 565.794,Z 512.346,A -85,B 0,C 180,E1 -10342.799,E2 -10342.799} C_VEL
LIN {X 0,Y 565.311,Z 522.189,A -85,B 0,C 180,E1 -10343.597,E2 -10343.597} C_VEL
LIN {X 0,Y 564.709,Z 533.019,A -85,B 0,C 180,E1 -10344.662,E2 -10344.662} C_VEL
LIN {X 0,Y 564.213,Z 541.957,A -85,B 0,C 180,E1 -10345.728,E2 -10345.728} C_VEL
LIN {X 0,Y 563.812,Z 550.491,A -85,B 0,C 180,E1 -10346.974,E2 -10346.974} C_VEL
LIN {X 0,Y 563.456,Z 557.398,A -85,B 0,C 180,E1 -10348.219,E2 -10348.219} C_VEL
LIN {X 0,Y 563.075,Z 563.62,A -85,B 0,C 180,E1 -10349.644,E2 -10349.644} C_VEL
LIN {X 0,Y 562.82,Z 567.217,A -85,B 0,C 180,E1 -10350.713,E2 -10350.713} C_VEL
LIN {X 0,Y 562.8,Z 570.722,A -85,B 0,C 180,E1 -10352.14,E2 -10352.14} C_VEL
LIN {X 0,Y 562.817,Z 572.879,A -85,B 0,C 180,E1 -10353.568,E2 -10353.568} C_VEL
LIN {X 0,Y 562.691,Z 573.76,A -85,B 0,C 180,E1 -10354.999,E2 -10354.999} C_VEL
LIN {X 0,Y 562.805,Z 573.33,A -85,B 0,C 180,E1 -10356.431,E2 -10356.431} C_VEL
LIN {X 0,Y 562.898,Z 571.608,A -85,B 0,C 180,E1 -10357.867,E2 -10357.867} C_VEL
LIN {X 0,Y 563.066,Z 568.533,A -85,B 0,C 180,E1 -10359.307,E2 -10359.307} C_VEL
LIN {X 0,Y 563.38,Z 565.221,A -85,B 0,C 180,E1 -10360.386,E2 -10360.386} C_VEL
LIN {X 0,Y 563.744,Z 559.487,A -85,B 0,C 180,E1 -10361.83,E2 -10361.83} C_VEL
LIN {X 0,Y 564.198,Z 552.995,A -85,B 0,C 180,E1 -10363.095,E2 -10363.095} C_VEL
LIN {X 0,Y 564.725,Z 544.882,A -85,B 0,C 180,E1 -10364.363,E2 -10364.363} C_VEL
LIN {X 0,Y 565.28,Z 536.369,A -85,B 0,C 180,E1 -10365.451,E2 -10365.451} C_VEL
LIN {X 0,Y 565.888,Z 526.008,A -85,B 0,C 180,E1 -10366.54,E2 -10366.54} C_VEL
LIN {X 0,Y 566.489,Z 514.851,A -85,B 0,C 180,E1 -10367.503,E2 -10367.503} C_VEL
LIN {X 0,Y 567.008,Z 504.075,A -85,B 0,C 180,E1 -10368.268,E2 -10368.268} C_VEL
LIN {X 0,Y 567.55,Z 491.439,A -85,B 0,C 180,E1 -10368.997,E2 -10368.997} C_VEL
LIN {X 0,Y 567.839,Z 478.301,A -85,B 0,C 180,E1 -10369.595,E2 -10369.595} C_VEL
LIN {X 0,Y 568.155,Z 464.795,A -85,B 0,C 180,E1 -10370.053,E2 -10370.053} C_VEL
LIN {X 0,Y 568.266,Z 451.282,A -85,B 0,C 180,E1 -10370.373,E2 -10370.373} C_VEL
LIN {X 0,Y 568.774,Z 395.906,A -85,B 0,C 180,E1 -10371.102,E2 -10371.102} C_VEL
LIN {X 0,Y 569.059,Z 343.177,A -85,B 0,C 180,E1 -10371.781,E2 -10371.781} C_VEL
LIN {X 0,Y 563.237,Z 327.892,A -85,B 0,C 180,E1 -10372.198,E2 -10372.198} C_VEL
LIN {X 0,Y 563.268,Z 327.884,A -85,B 0,C 180,E1 -10375.012,E2 -10375.012} C_VEL
LIN {X 0,Y 563.261,Z 327.881,A -85,B 0,C 180,E1 -10378.2,E2 -10378.2} C_VEL
LIN {X 0,Y 563.233,Z 327.882,A -85,B 0,C 180,E1 -10380.896,E2 -10380.896} C_VEL
LIN {X 0,Y 563.213,Z 327.884,A -85,B 0,C 180,E1 -10383.565,E2 -10383.565} C_VEL
LIN {X 0,Y 563.232,Z 327.884,A -85,B 0,C 180,E1 -10386.651,E2 -10386.651} C_VEL
LIN {X 0,Y 563.23,Z 327.882,A -85,B 0,C 180,E1 -10389.552,E2 -10389.552} C_VEL
LIN {X 0,Y 563.216,Z 327.889,A -85,B 0,C 180,E1 -10392.189,E2 -10392.189} C_VEL
LIN {X 0,Y 563.275,Z 327.873,A -85,B 0,C 180,E1 -10395.138,E2 -10395.138} C_VEL
LIN {X 0,Y 563.266,Z 327.881,A -85,B 0,C 180,E1 -10397.816,E2 -10397.816} C_VEL
LIN {X 0,Y 563.216,Z 327.88,A -85,B 0,C 180,E1 -10400.634,E2 -10400.634} C_VEL
LIN {X 0,Y 563.253,Z 327.863,A -85,B 0,C 180,E1 -10403.933,E2 -10403.933} C_VEL
LIN {X 0,Y 563.225,Z 327.879,A -85,B 0,C 180,E1 -10406.825,E2 -10406.825} C_VEL
LIN {X 0,Y 563.246,Z 327.876,A -85,B 0,C 180,E1 -10409.344,E2 -10409.344} C_VEL
LIN {X 0,Y 563.266,Z 327.88,A -85,B 0,C 180,E1 -10411.997,E2 -10411.997} C_VEL
LIN {X 0,Y 563.264,Z 327.874,A -85,B 0,C 180,E1 -10415.202,E2 -10415.202} C_VEL
LIN {X 0,Y 563.229,Z 327.879,A -85,B 0,C 180,E1 -10418.094,E2 -10418.094} C_VEL
LIN {X 0,Y 563.29,Z 327.879,A -85,B 0,C 180,E1 -10421.137,E2 -10421.137} C_VEL
LIN {X 0,Y 563.272,Z 327.882,A -85,B 0,C 180,E1 -10422.589,E2 -10422.589} C_VEL
LIN {X 0,Y 567.361,Z 341.296,A -85,B 0,C 180,E1 -10422.903,E2 -10422.903} C_VEL
LIN {X 0,Y 566.19,Z 448.752,A -85,B 0,C 180,E1 -10424.485,E2 -10424.485} C_VEL
LIN {X 0,Y 566.046,Z 464.033,A -85,B 0,C 180,E1 -10424.87,E2 -10424.87} C_VEL
LIN {X 0,Y 565.78,Z 478.478,A -85,B 0,C 180,E1 -10425.389,E2 -10425.389} C_VEL
LIN {X 0,Y 565.439,Z 491.745,A -85,B 0,C 180,E1 -10426.021,E2 -10426.021} C_VEL
LIN {X 0,Y 565.081,Z 503.851,A -85,B 0,C 180,E1 -10426.743,E2 -10426.743} C_VEL
LIN {X 0,Y 564.632,Z 516.156,A -85,B 0,C 180,E1 -10427.643,E2 -10427.643} C_VEL
LIN {X 0,Y 564.208,Z 527.44,A -85,B 0,C 180,E1 -10428.651,E2 -10428.651} C_VEL
LIN {X 0,Y 563.956,Z 536.444,A -85,B 0,C 180,E1 -10429.625,E2 -10429.625} C_VEL
LIN {X 0,Y 563.55,Z 544.808,A -85,B 0,C 180,E1 -10430.701,E2 -10430.701} C_VEL
LIN {X 0,Y 563.243,Z 552.775,A -85,B 0,C 180,E1 -10431.957,E2 -10431.957} C_VEL
LIN {X 0,Y 563.023,Z 559.177,A -85,B 0,C 180,E1 -10433.212,E2 -10433.212} C_VEL
LIN {X 0,Y 562.865,Z 563.581,A -85,B 0,C 180,E1 -10434.286,E2 -10434.286} C_VEL
LIN {X 0,Y 562.707,Z 568.013,A -85,B 0,C 180,E1 -10435.717,E2 -10435.717} C_VEL
LIN {X 0,Y 562.795,Z 569.657,A -85,B 0,C 180,E1 -10436.432,E2 -10436.432} C_VEL
LIN {X 0,Y 562.723,Z 571.909,A -85,B 0,C 180,E1 -10437.86,E2 -10437.86} C_VEL
LIN {X 0,Y 562.553,Z 572.766,A -85,B 0,C 180,E1 -10439.286,E2 -10439.286} C_VEL
LIN {X 0,Y 562.571,Z 572.208,A -85,B 0,C 180,E1 -10440.713,E2 -10440.713} C_VEL
LIN {X 0,Y 562.788,Z 570.252,A -85,B 0,C 180,E1 -10442.14,E2 -10442.14} C_VEL
LIN {X 0,Y 563.212,Z 566.853,A -85,B 0,C 180,E1 -10443.565,E2 -10443.565} C_VEL
LIN {X 0,Y 563.412,Z 563.298,A -85,B 0,C 180,E1 -10444.635,E2 -10444.635} C_VEL
LIN {X 0,Y 563.456,Z 558.85,A -85,B 0,C 180,E1 -10445.707,E2 -10445.707} C_VEL
LIN {X 0,Y 564.048,Z 552.255,A -85,B 0,C 180,E1 -10446.954,E2 -10446.954} C_VEL
LIN {X 0,Y 564.476,Z 544.089,A -85,B 0,C 180,E1 -10448.204,E2 -10448.204} C_VEL
LIN {X 0,Y 564.908,Z 535.512,A -85,B 0,C 180,E1 -10449.276,E2 -10449.276} C_VEL
LIN {X 0,Y 565.313,Z 526.951,A -85,B 0,C 180,E1 -10450.169,E2 -10450.169} C_VEL
LIN {X 0,Y 565.78,Z 516.769,A -85,B 0,C 180,E1 -10451.063,E2 -10451.063} C_VEL
LIN {X 0,Y 566.313,Z 505.697,A -85,B 0,C 180,E1 -10451.866,E2 -10451.866} C_VEL
LIN {X 0,Y 566.853,Z 492.632,A -85,B 0,C 180,E1 -10452.631,E2 -10452.631} C_VEL
LIN {X 0,Y 567.134,Z 479.219,A -85,B 0,C 180,E1 -10453.253,E2 -10453.253} C_VEL
LIN {X 0,Y 567.369,Z 465.069,A -85,B 0,C 180,E1 -10453.748,E2 -10453.748} C_VEL
LIN {X 0,Y 567.56,Z 450.972,A -85,B 0,C 180,E1 -10454.085,E2 -10454.085} C_VEL
LIN {X 0,Y 569.133,Z 354.507,A -85,B 0,C 180,E1 -10455.609,E2 -10455.609} C_VEL
LIN {X 0,Y 569.241,Z 342.747,A -85,B 0,C 180,E1 -10455.806,E2 -10455.806} C_VEL
LIN {X 0,Y 563.453,Z 328.552,A -85,B 0,C 180,E1 -10456.311,E2 -10456.311} C_VEL
LIN {X 0,Y 563.337,Z 327.875,A -85,B 0,C 180,E1 -10456.335,E2 -10456.335} C_VEL
LIN {X 0,Y 563.297,Z 327.877,A -85,B 0,C 180,E1 -10459.083,E2 -10459.083} C_VEL
LIN {X 0,Y 563.301,Z 327.879,A -85,B 0,C 180,E1 -10461.903,E2 -10461.903} C_VEL
LIN {X 0,Y 563.266,Z 327.879,A -85,B 0,C 180,E1 -10464.798,E2 -10464.798} C_VEL
LIN {X 0,Y 563.294,Z 327.881,A -85,B 0,C 180,E1 -10468.009,E2 -10468.009} C_VEL
LIN {X 0,Y 563.251,Z 327.879,A -85,B 0,C 180,E1 -10470.899,E2 -10470.899} C_VEL
LIN {X 0,Y 563.258,Z 327.88,A -85,B 0,C 180,E1 -10473.572,E2 -10473.572} C_VEL
LIN {X 0,Y 563.327,Z 327.867,A -85,B 0,C 180,E1 -10476.078,E2 -10476.078} C_VEL
LIN {X 0,Y 563.239,Z 327.875,A -85,B 0,C 180,E1 -10478.448,E2 -10478.448} C_VEL
LIN {X 0,Y 563.235,Z 327.882,A -85,B 0,C 180,E1 -10481.232,E2 -10481.232} C_VEL
LIN {X 0,Y 563.251,Z 327.875,A -85,B 0,C 180,E1 -10484.139,E2 -10484.139} C_VEL
LIN {X 0,Y 563.257,Z 327.882,A -85,B 0,C 180,E1 -10487.197,E2 -10487.197} C_VEL
LIN {X 0,Y 563.236,Z 327.88,A -85,B 0,C 180,E1 -10489.708,E2 -10489.708} C_VEL
LIN {X 0,Y 563.207,Z 327.89,A -85,B 0,C 180,E1 -10492.745,E2 -10492.745} C_VEL
LIN {X 0,Y 563.214,Z 327.88,A -85,B 0,C 180,E1 -10495.166,E2 -10495.166} C_VEL
LIN {X 0,Y 563.241,Z 327.882,A -85,B 0,C 180,E1 -10497.741,E2 -10497.741} C_VEL
LIN {X 0,Y 563.248,Z 327.885,A -85,B 0,C 180,E1 -10500.518,E2 -10500.518} C_VEL
LIN {X 0,Y 563.308,Z 328.039,A -85,B 0,C 180,E1 -10501.019,E2 -10501.019} C_VEL
LIN {X 0,Y 567.106,Z 345.3,A -85,B 0,C 180,E1 -10503.237,E2 -10503.237} C_VEL
LIN {X 0,Y 567.582,Z 350.126,A -85,B 0,C 180,E1 -10503.82,E2 -10503.82} C_VEL
LIN {X 0,Y 566.652,Z 368.576,A -85,B 0,C 180,E1 -10505.926,E2 -10505.926} C_VEL
LIN {X 0,Y 565.443,Z 395.347,A -85,B 0,C 180,E1 -10508.946,E2 -10508.946} C_VEL
LIN {X 0,Y 564.446,Z 420.341,A -85,B 0,C 180,E1 -10511.739,E2 -10511.739} C_VEL
LIN {X 0,Y 564.18,Z 429.447,A -85,B 0,C 180,E1 -10512.753,E2 -10512.753} C_VEL
LIN {X 0,Y 567.628,Z 458.458,A -85,B 0,C 180,E1 -10513.245,E2 -10513.245} C_VEL
LIN {X 0,Y 568.205,Z 466.953,A -85,B 0,C 180,E1 -10513.374,E2 -10513.374} C_VEL
LIN {X 0,Y 567.22,Z 568.81,A -85,B 0,C 180,E1 -10514.68,E2 -10514.68} C_VEL
LIN {X 0,Y 566.701,Z 583.245,A -85,B 0,C 180,E1 -10515.002,E2 -10515.002} C_VEL
LIN {X 0,Y 566.066,Z 596.764,A -85,B 0,C 180,E1 -10515.443,E2 -10515.443} C_VEL
LIN {X 0,Y 565.383,Z 609.984,A -85,B 0,C 180,E1 -10516.02,E2 -10516.02} C_VEL
LIN {X 0,Y 564.74,Z 622.779,A -85,B 0,C 180,E1 -10516.735,E2 -10516.735} C_VEL
LIN {X 0,Y 563.745,Z 644.642,A -85,B 0,C 180,E1 -10518.17,E2 -10518.17} C_VEL
LIN {X 0,Y 563.35,Z 656.177,A -85,B 0,C 180,E1 -10519.104,E2 -10519.104} C_VEL
LIN {X 0,Y 562.892,Z 666.776,A -85,B 0,C 180,E1 -10520.148,E2 -10520.148} C_VEL
LIN {X 0,Y 562.612,Z 675.817,A -85,B 0,C 180,E1 -10521.227,E2 -10521.227} C_VEL
LIN {X 0,Y 562.376,Z 683.301,A -85,B 0,C 180,E1 -10522.305,E2 -10522.305} C_VEL
LIN {X 0,Y 562.214,Z 690.425,A -85,B 0,C 180,E1 -10523.562,E2 -10523.562} C_VEL
LIN {X 0,Y 562.163,Z 695.316,A -85,B 0,C 180,E1 -10524.638,E2 -10524.638} C_VEL
LIN {X 0,Y 562.003,Z 699.889,A -85,B 0,C 180,E1 -10525.924,E2 -10525.924} C_VEL
LIN {X 0,Y 562.026,Z 703.03,A -85,B 0,C 180,E1 -10527.142,E2 -10527.142} C_VEL
LIN {X 0,Y 561.968,Z 705.338,A -85,B 0,C 180,E1 -10528.571,E2 -10528.571} C_VEL
LIN {X 0,Y 561.957,Z 706.212,A -85,B 0,C 180,E1 -10530,E2 -10530} C_VEL
LIN {X 0,Y 561.967,Z 705.662,A -85,B 0,C 180,E1 -10531.428,E2 -10531.428} C_VEL
LIN {X 0,Y 562.047,Z 703.663,A -85,B 0,C 180,E1 -10532.857,E2 -10532.857} C_VEL
LIN {X 0,Y 562.057,Z 700.169,A -85,B 0,C 180,E1 -10534.288,E2 -10534.288} C_VEL
LIN {X 0,Y 562.194,Z 695.101,A -85,B 0,C 180,E1 -10535.72,E2 -10535.72} C_VEL
LIN {X 0,Y 562.315,Z 690.169,A -85,B 0,C 180,E1 -10536.796,E2 -10536.796} C_VEL
LIN {X 0,Y 562.588,Z 683.009,A -85,B 0,C 180,E1 -10538.052,E2 -10538.052} C_VEL
LIN {X 0,Y 562.847,Z 675.51,A -85,B 0,C 180,E1 -10539.13,E2 -10539.13} C_VEL
LIN {X 0,Y 563.26,Z 666.467,A -85,B 0,C 180,E1 -10540.207,E2 -10540.207} C_VEL
LIN {X 0,Y 563.662,Z 657.47,A -85,B 0,C 180,E1 -10541.105,E2 -10541.105} C_VEL
LIN {X 0,Y 564.188,Z 645.537,A -85,B 0,C 180,E1 -10542.093,E2 -10542.093} C_VEL
LIN {X 0,Y 564.688,Z 633.596,A -85,B 0,C 180,E1 -10542.901,E2 -10542.901} C_VEL
LIN {X 0,Y 565.281,Z 620.372,A -85,B 0,C 180,E1 -10543.617,E2 -10543.617} C_VEL
LIN {X 0,Y 565.742,Z 606.489,A -85,B 0,C 180,E1 -10544.199,E2 -10544.199} C_VEL
LIN {X 0,Y 566.13,Z 592.014,A -85,B 0,C 180,E1 -10544.647,E2 -10544.647} C_VEL
LIN {X 0,Y 566.478,Z 577.943,A -85,B 0,C 180,E1 -10544.935,E2 -10544.935} C_VEL
LIN {X 0,Y 568.306,Z 477.102,A -85,B 0,C 180,E1 -10546.532,E2 -10546.532} C_VEL
LIN {X 0,Y 568.33,Z 462.308,A -85,B 0,C 180,E1 -10546.789,E2 -10546.789} C_VEL
LIN {X 0,Y 566.145,Z 438.837,A -85,B 0,C 180,E1 -10547.298,E2 -10547.298} C_VEL
LIN {X 0,Y 565.177,Z 430.676,A -85,B 0,C 180,E1 -10547.533,E2 -10547.533} C_VEL
LIN {X 0,Y 564.083,Z 420.975,A -85,B 0,C 180,E1 -10547.875,E2 -10547.875} C_VEL
LIN {X 0,Y 564.901,Z 397.041,A -85,B 0,C 180,E1 -10550.505,E2 -10550.505} C_VEL
LIN {X 0,Y 565.736,Z 374.882,A -85,B 0,C 180,E1 -10552.955,E2 -10552.955} C_VEL
LIN {X 0,Y 566.781,Z 349.144,A -85,B 0,C 180,E1 -10555.825,E2 -10555.825} C_VEL
LIN {X 0,Y 566.547,Z 343.914,A -85,B 0,C 180,E1 -10556.429,E2 -10556.429} C_VEL
LIN {X 0,Y 563.265,Z 327.882,A -85,B 0,C 180,E1 -10558.402,E2 -10558.402} C_VEL
LIN {X 0,Y 563.244,Z 327.886,A -85,B 0,C 180,E1 -10561.487,E2 -10561.487} C_VEL
LIN {X 0,Y 563.216,Z 327.884,A -85,B 0,C 180,E1 -10564.031,E2 -10564.031} C_VEL
LIN {X 0,Y 563.219,Z 327.884,A -85,B 0,C 180,E1 -10566.652,E2 -10566.652} C_VEL
LIN {X 0,Y 563.223,Z 327.883,A -85,B 0,C 180,E1 -10569.551,E2 -10569.551} C_VEL
LIN {X 0,Y 563.211,Z 327.885,A -85,B 0,C 180,E1 -10572.189,E2 -10572.189} C_VEL
LIN {X 0,Y 563.27,Z 327.884,A -85,B 0,C 180,E1 -10575.138,E2 -10575.138} C_VEL
LIN {X 0,Y 563.205,Z 327.887,A -85,B 0,C 180,E1 -10578.263,E2 -10578.263} C_VEL
LIN {X 0,Y 563.213,Z 327.886,A -85,B 0,C 180,E1 -10580.635,E2 -10580.635} C_VEL
LIN {X 0,Y 563.284,Z 327.878,A -85,B 0,C 180,E1 -10583.928,E2 -10583.928} C_VEL
LIN {X 0,Y 563.225,Z 327.89,A -85,B 0,C 180,E1 -10586.825,E2 -10586.825} C_VEL
LIN {X 0,Y 563.253,Z 327.891,A -85,B 0,C 180,E1 -10589.345,E2 -10589.345} C_VEL
LIN {X 0,Y 563.245,Z 327.903,A -85,B 0,C 180,E1 -10590.429,E2 -10590.429} C_VEL
LIN {X 0,Y 567.27,Z 341.772,A -85,B 0,C 180,E1 -10592.206,E2 -10592.206} C_VEL
LIN {X 0,Y 569.262,Z 350.932,A -85,B 0,C 180,E1 -10593.313,E2 -10593.313} C_VEL
LIN {X 0,Y 569.29,Z 356.576,A -85,B 0,C 180,E1 -10593.92,E2 -10593.92} C_VEL
LIN {X 0,Y 568.215,Z 383.644,A -85,B 0,C 180,E1 -10596.767,E2 -10596.767} C_VEL
LIN {X 0,Y 567.212,Z 408.84,A -85,B 0,C 180,E1 -10599.394,E2 -10599.394} C_VEL
LIN {X 0,Y 566.297,Z 436.092,A -85,B 0,C 180,E1 -10602.251,E2 -10602.251} C_VEL
LIN {X 0,Y 566.172,Z 439.626,A -85,B 0,C 180,E1 -10602.621,E2 -10602.621} C_VEL
LIN {X 0,Y 568.771,Z 457.209,A -85,B 0,C 180,E1 -10603.04,E2 -10603.04} C_VEL
LIN {X 0,Y 569.134,Z 462.297,A -85,B 0,C 180,E1 -10603.143,E2 -10603.143} C_VEL
LIN {X 0,Y 567.22,Z 563.606,A -85,B 0,C 180,E1 -10604.744,E2 -10604.744} C_VEL
LIN {X 0,Y 566.834,Z 583.057,A -85,B 0,C 180,E1 -10605.074,E2 -10605.074} C_VEL
LIN {X 0,Y 566.405,Z 597.03,A -85,B 0,C 180,E1 -10605.452,E2 -10605.452} C_VEL
LIN {X 0,Y 565.922,Z 610.232,A -85,B 0,C 180,E1 -10605.942,E2 -10605.942} C_VEL
LIN {X 0,Y 565.409,Z 623.258,A -85,B 0,C 180,E1 -10606.569,E2 -10606.569} C_VEL
LIN {X 0,Y 564.802,Z 635.212,A -85,B 0,C 180,E1 -10607.284,E2 -10607.284} C_VEL
LIN {X 0,Y 564.197,Z 647.447,A -85,B 0,C 180,E1 -10608.18,E2 -10608.18} C_VEL
LIN {X 0,Y 563.67,Z 658.498,A -85,B 0,C 180,E1 -10609.173,E2 -10609.173} C_VEL
LIN {X 0,Y 563.264,Z 667.597,A -85,B 0,C 180,E1 -10610.155,E2 -10610.155} C_VEL
LIN {X 0,Y 562.839,Z 675.946,A -85,B 0,C 180,E1 -10611.231,E2 -10611.231} C_VEL
LIN {X 0,Y 562.502,Z 683.922,A -85,B 0,C 180,E1 -10612.487,E2 -10612.487} C_VEL
LIN {X 0,Y 562.296,Z 689.519,A -85,B 0,C 180,E1 -10613.563,E2 -10613.563} C_VEL
LIN {X 0,Y 562.073,Z 695.362,A -85,B 0,C 180,E1 -10614.996,E2 -10614.996} C_VEL
LIN {X 0,Y 561.996,Z 699.596,A -85,B 0,C 180,E1 -10616.427,E2 -10616.427} C_VEL
LIN {X 0,Y 561.921,Z 702.337,A -85,B 0,C 180,E1 -10617.857,E2 -10617.857} C_VEL
LIN {X 0,Y 561.864,Z 703.63,A -85,B 0,C 180,E1 -10619.286,E2 -10619.286} C_VEL
LIN {X 0,Y 561.863,Z 703.504,A -85,B 0,C 180,E1 -10620.714,E2 -10620.714} C_VEL
LIN {X 0,Y 561.919,Z 701.973,A -85,B 0,C 180,E1 -10622.143,E2 -10622.143} C_VEL
LIN {X 0,Y 561.973,Z 699.015,A -85,B 0,C 180,E1 -10623.573,E2 -10623.573} C_VEL
LIN {X 0,Y 562.077,Z 694.554,A -85,B 0,C 180,E1 -10625.005,E2 -10625.005} C_VEL
LIN {X 0,Y 562.161,Z 690.092,A -85,B 0,C 180,E1 -10626.08,E2 -10626.08} C_VEL
LIN {X 0,Y 562.37,Z 683.606,A -85,B 0,C 180,E1 -10627.335,E2 -10627.335} C_VEL
LIN {X 0,Y 562.606,Z 675.527,A -85,B 0,C 180,E1 -10628.592,E2 -10628.592} C_VEL
LIN {X 0,Y 563.012,Z 667.056,A -85,B 0,C 180,E1 -10629.669,E2 -10629.669} C_VEL
LIN {X 0,Y 563.413,Z 656.788,A -85,B 0,C 180,E1 -10630.748,E2 -10630.748} C_VEL
LIN {X 0,Y 563.831,Z 645.332,A -85,B 0,C 180,E1 -10631.738,E2 -10631.738} C_VEL
LIN {X 0,Y 564.372,Z 632.582,A -85,B 0,C 180,E1 -10632.636,E2 -10632.636} C_VEL
LIN {X 0,Y 564.914,Z 619.939,A -85,B 0,C 180,E1 -10633.352,E2 -10633.352} C_VEL
LIN {X 0,Y 565.405,Z 606.93,A -85,B 0,C 180,E1 -10633.934,E2 -10633.934} C_VEL
LIN {X 0,Y 565.71,Z 592.995,A -85,B 0,C 180,E1 -10634.406,E2 -10634.406} C_VEL
LIN {X 0,Y 566.022,Z 578.774,A -85,B 0,C 180,E1 -10634.742,E2 -10634.742} C_VEL
LIN {X 0,Y 567.481,Z 458.269,A -85,B 0,C 180,E1 -10636.522,E2 -10636.522} C_VEL
LIN {X 0,Y 565.183,Z 439.444,A -85,B 0,C 180,E1 -10636.886,E2 -10636.886} C_VEL
LIN {X 0,Y 566.155,Z 408.513,A -85,B 0,C 180,E1 -10640.139,E2 -10640.139} C_VEL
LIN {X 0,Y 567.193,Z 378.789,A -85,B 0,C 180,E1 -10643.277,E2 -10643.277} C_VEL
LIN {X 0,Y 568.131,Z 351.496,A -85,B 0,C 180,E1 -10646.169,E2 -10646.169} C_VEL
LIN {X 0,Y 567.839,Z 347.978,A -85,B 0,C 180,E1 -10646.557,E2 -10646.557} C_VEL
LIN {X 0,Y 563.332,Z 327.874,A -85,B 0,C 180,E1 -10648.924,E2 -10648.924} C_VEL
LIN {X 0,Y 563.286,Z 327.88,A -85,B 0,C 180,E1 -10651.485,E2 -10651.485} C_VEL
LIN {X 0,Y 563.267,Z 327.875,A -85,B 0,C 180,E1 -10654.028,E2 -10654.028} C_VEL
LIN {X 0,Y 563.281,Z 327.875,A -85,B 0,C 180,E1 -10656.647,E2 -10656.647} C_VEL
LIN {X 0,Y 563.261,Z 327.878,A -85,B 0,C 180,E1 -10659.556,E2 -10659.556} C_VEL
LIN {X 0,Y 563.273,Z 327.874,A -85,B 0,C 180,E1 -10662.184,E2 -10662.184} C_VEL
LIN {X 0,Y 563.275,Z 327.88,A -85,B 0,C 180,E1 -10665.138,E2 -10665.138} C_VEL
LIN {X 0,Y 563.273,Z 327.874,A -85,B 0,C 180,E1 -10667.817,E2 -10667.817} C_VEL
LIN {X 0,Y 563.225,Z 327.888,A -85,B 0,C 180,E1 -10670.635,E2 -10670.635} C_VEL
LIN {X 0,Y 563.328,Z 327.868,A -85,B 0,C 180,E1 -10673.922,E2 -10673.922} C_VEL
LIN {X 0,Y 563.258,Z 327.881,A -85,B 0,C 180,E1 -10676.827,E2 -10676.827} C_VEL
LIN {X 0,Y 563.265,Z 327.876,A -85,B 0,C 180,E1 -10679.346,E2 -10679.346} C_VEL
LIN {X 0,Y 563.294,Z 327.875,A -85,B 0,C 180,E1 -10681.991,E2 -10681.991} C_VEL
LIN {X 0,Y 563.222,Z 327.885,A -85,B 0,C 180,E1 -10684.436,E2 -10684.436} C_VEL
LIN {X 0,Y 562.579,Z 327.963,A -85,B 0,C 180,E1 -10685.033,E2 -10685.033} C_VEL
LIN {X 0,Y 559.739,Z 328.32,A -85,B 0,C 180,E1 -10686.002,E2 -10686.002} C_VEL
LIN {X 0,Y 557.333,Z 328.616,A -85,B 0,C 180,E1 -10686.783,E2 -10686.783} C_VEL
LIN {X 0,Y 556.31,Z 328.742,A -85,B 0,C 180,E1 -10687.385,E2 -10687.385} C_VEL
LIN {X 0,Y 556.233,Z 328.753,A -85,B 0,C 180,E1 -10687.589,E2 -10687.589} C_VEL
LIN {X 0,Y 556.243,Z 328.759,A -85,B 0,C 180,E1 -10690.123,E2 -10690.123} C_VEL
LIN {X 0,Y 556.269,Z 328.748,A -85,B 0,C 180,E1 -10693.165,E2 -10693.165} C_VEL
LIN {X 0,Y 556.316,Z 328.746,A -85,B 0,C 180,E1 -10696.159,E2 -10696.159} C_VEL
LIN {X 0,Y 556.293,Z 328.75,A -85,B 0,C 180,E1 -10698.2,E2 -10698.2} C_VEL
LIN {X 0,Y 561.055,Z 342.874,A -85,B 0,C 180,E1 -10698.529,E2 -10698.529} C_VEL
LIN {X 0,Y 560.412,Z 447.235,A -85,B 0,C 180,E1 -10699.877,E2 -10699.877} C_VEL
LIN {X 0,Y 560.292,Z 461.486,A -85,B 0,C 180,E1 -10700.17,E2 -10700.17} C_VEL
LIN {X 0,Y 560.087,Z 475.205,A -85,B 0,C 180,E1 -10700.598,E2 -10700.598} C_VEL
LIN {X 0,Y 559.708,Z 488.971,A -85,B 0,C 180,E1 -10701.182,E2 -10701.182} C_VEL
LIN {X 0,Y 559.306,Z 502.052,A -85,B 0,C 180,E1 -10701.908,E2 -10701.908} C_VEL
LIN {X 0,Y 558.859,Z 513.662,A -85,B 0,C 180,E1 -10702.71,E2 -10702.71} C_VEL
LIN {X 0,Y 558.346,Z 523.425,A -85,B 0,C 180,E1 -10703.517,E2 -10703.517} C_VEL
LIN {X 0,Y 557.71,Z 534.169,A -85,B 0,C 180,E1 -10704.595,E2 -10704.595} C_VEL
LIN {X 0,Y 557.207,Z 543.042,A -85,B 0,C 180,E1 -10705.675,E2 -10705.675} C_VEL
LIN {X 0,Y 556.787,Z 551.519,A -85,B 0,C 180,E1 -10706.935,E2 -10706.935} C_VEL
LIN {X 0,Y 556.411,Z 558.379,A -85,B 0,C 180,E1 -10708.197,E2 -10708.197} C_VEL
LIN {X 0,Y 556.034,Z 564.554,A -85,B 0,C 180,E1 -10709.639,E2 -10709.639} C_VEL
LIN {X 0,Y 555.768,Z 568.109,A -85,B 0,C 180,E1 -10710.722,E2 -10710.722} C_VEL
LIN {X 0,Y 555.77,Z 571.572,A -85,B 0,C 180,E1 -10712.167,E2 -10712.167} C_VEL
LIN {X 0,Y 555.756,Z 573.695,A -85,B 0,C 180,E1 -10713.613,E2 -10713.613} C_VEL
LIN {X 0,Y 555.651,Z 574.536,A -85,B 0,C 180,E1 -10715.063,E2 -10715.063} C_VEL
LIN {X 0,Y 555.754,Z 574.071,A -85,B 0,C 180,E1 -10716.513,E2 -10716.513} C_VEL
LIN {X 0,Y 555.879,Z 572.309,A -85,B 0,C 180,E1 -10717.967,E2 -10717.967} C_VEL
LIN {X 0,Y 556.062,Z 569.186,A -85,B 0,C 180,E1 -10719.425,E2 -10719.425} C_VEL
LIN {X 0,Y 556.448,Z 564.558,A -85,B 0,C 180,E1 -10720.884,E2 -10720.884} C_VEL
LIN {X 0,Y 556.904,Z 558.312,A -85,B 0,C 180,E1 -10722.346,E2 -10722.346} C_VEL
LIN {X 0,Y 557.381,Z 551.33,A -85,B 0,C 180,E1 -10723.629,E2 -10723.629} C_VEL
LIN {X 0,Y 557.969,Z 543.141,A -85,B 0,C 180,E1 -10724.845,E2 -10724.845} C_VEL
LIN {X 0,Y 558.625,Z 533.524,A -85,B 0,C 180,E1 -10726.013,E2 -10726.013} C_VEL
LIN {X 0,Y 559.216,Z 523.395,A -85,B 0,C 180,E1 -10727.025,E2 -10727.025} C_VEL
LIN {X 0,Y 559.774,Z 512.083,A -85,B 0,C 180,E1 -10727.954,E2 -10727.954} C_VEL
LIN {X 0,Y 560.434,Z 499.717,A -85,B 0,C 180,E1 -10728.774,E2 -10728.774} C_VEL
LIN {X 0,Y 560.918,Z 487.61,A -85,B 0,C 180,E1 -10729.419,E2 -10729.419} C_VEL
LIN {X 0,Y 561.176,Z 475.518,A -85,B 0,C 180,E1 -10729.932,E2 -10729.932} C_VEL
LIN {X 0,Y 561.436,Z 461.324,A -85,B 0,C 180,E1 -10730.375,E2 -10730.375} C_VEL
LIN {X 0,Y 561.556,Z 447.496,A -85,B 0,C 180,E1 -10730.659,E2 -10730.659} C_VEL
LIN {X 0,Y 562.372,Z 344.862,A -85,B 0,C 180,E1 -10731.996,E2 -10731.996} C_VEL
LIN {X 0,Y 556.191,Z 328.77,A -85,B 0,C 180,E1 -10732.443,E2 -10732.443} C_VEL
LIN {X 0,Y 556.208,Z 328.762,A -85,B 0,C 180,E1 -10735.352,E2 -10735.352} C_VEL
LIN {X 0,Y 556.23,Z 328.757,A -85,B 0,C 180,E1 -10738.177,E2 -10738.177} C_VEL
LIN {X 0,Y 556.206,Z 328.756,A -85,B 0,C 180,E1 -10741.091,E2 -10741.091} C_VEL
LIN {X 0,Y 556.18,Z 328.762,A -85,B 0,C 180,E1 -10743.778,E2 -10743.778} C_VEL
LIN {X 0,Y 556.209,Z 328.762,A -85,B 0,C 180,E1 -10746.296,E2 -10746.296} C_VEL
LIN {X 0,Y 556.153,Z 328.763,A -85,B 0,C 180,E1 -10749.03,E2 -10749.03} C_VEL
LIN {X 0,Y 556.199,Z 328.758,A -85,B 0,C 180,E1 -10750.921,E2 -10750.921} C_VEL
LIN {X 0,Y 556.228,Z 328.759,A -85,B 0,C 180,E1 -10754.127,E2 -10754.127} C_VEL
LIN {X 0,Y 556.226,Z 328.753,A -85,B 0,C 180,E1 -10756.919,E2 -10756.919} C_VEL
LIN {X 0,Y 556.184,Z 328.764,A -85,B 0,C 180,E1 -10760.037,E2 -10760.037} C_VEL
LIN {X 0,Y 556.163,Z 328.742,A -85,B 0,C 180,E1 -10762.805,E2 -10762.805} C_VEL
LIN {X 0,Y 556.194,Z 328.75,A -85,B 0,C 180,E1 -10765.479,E2 -10765.479} C_VEL
LIN {X 0,Y 556.203,Z 328.757,A -85,B 0,C 180,E1 -10768.067,E2 -10768.067} C_VEL
LIN {X 0,Y 556.223,Z 328.751,A -85,B 0,C 180,E1 -10770.585,E2 -10770.585} C_VEL
LIN {X 0,Y 556.221,Z 328.755,A -85,B 0,C 180,E1 -10773.393,E2 -10773.393} C_VEL
LIN {X 0,Y 556.203,Z 328.757,A -85,B 0,C 180,E1 -10776.235,E2 -10776.235} C_VEL
LIN {X 0,Y 556.196,Z 328.756,A -85,B 0,C 180,E1 -10779.352,E2 -10779.352} C_VEL
LIN {X 0,Y 556.232,Z 328.765,A -85,B 0,C 180,E1 -10781.65,E2 -10781.65} C_VEL
LIN {X 0,Y 556.226,Z 328.761,A -85,B 0,C 180,E1 -10782.431,E2 -10782.431} C_VEL
LIN {X 0,Y 560.455,Z 342.274,A -85,B 0,C 180,E1 -10782.75,E2 -10782.75} C_VEL
LIN {X 0,Y 559.252,Z 448.577,A -85,B 0,C 180,E1 -10784.339,E2 -10784.339} C_VEL
LIN {X 0,Y 559.057,Z 463.554,A -85,B 0,C 180,E1 -10784.711,E2 -10784.711} C_VEL
LIN {X 0,Y 558.829,Z 478.023,A -85,B 0,C 180,E1 -10785.227,E2 -10785.227} C_VEL
LIN {X 0,Y 558.493,Z 491.192,A -85,B 0,C 180,E1 -10785.844,E2 -10785.844} C_VEL
LIN {X 0,Y 558.134,Z 503.543,A -85,B 0,C 180,E1 -10786.575,E2 -10786.575} C_VEL
LIN {X 0,Y 557.681,Z 516.03,A -85,B 0,C 180,E1 -10787.487,E2 -10787.487} C_VEL
LIN {X 0,Y 557.253,Z 526.333,A -85,B 0,C 180,E1 -10788.398,E2 -10788.398} C_VEL
LIN {X 0,Y 556.961,Z 536.605,A -85,B 0,C 180,E1 -10789.493,E2 -10789.493} C_VEL
LIN {X 0,Y 556.533,Z 545.097,A -85,B 0,C 180,E1 -10790.583,E2 -10790.583} C_VEL
LIN {X 0,Y 556.213,Z 553.178,A -85,B 0,C 180,E1 -10791.855,E2 -10791.855} C_VEL
LIN {X 0,Y 555.987,Z 559.665,A -85,B 0,C 180,E1 -10793.126,E2 -10793.126} C_VEL
LIN {X 0,Y 555.821,Z 564.142,A -85,B 0,C 180,E1 -10794.214,E2 -10794.214} C_VEL
LIN {X 0,Y 555.649,Z 568.647,A -85,B 0,C 180,E1 -10795.662,E2 -10795.662} C_VEL
LIN {X 0,Y 555.697,Z 571.656,A -85,B 0,C 180,E1 -10797.11,E2 -10797.11} C_VEL
LIN {X 0,Y 555.592,Z 573.285,A -85,B 0,C 180,E1 -10798.555,E2 -10798.555} C_VEL
LIN {X 0,Y 555.498,Z 573.505,A -85,B 0,C 180,E1 -10800,E2 -10800} C_VEL
LIN {X 0,Y 555.616,Z 572.303,A -85,B 0,C 180,E1 -10801.445,E2 -10801.445} C_VEL
LIN {X 0,Y 555.982,Z 569.676,A -85,B 0,C 180,E1 -10802.888,E2 -10802.888} C_VEL
LIN {X 0,Y 556.423,Z 565.585,A -85,B 0,C 180,E1 -10804.332,E2 -10804.332} C_VEL
LIN {X 0,Y 556.406,Z 561.491,A -85,B 0,C 180,E1 -10805.418,E2 -10805.418} C_VEL
LIN {X 0,Y 556.885,Z 556.351,A -85,B 0,C 180,E1 -10806.5,E2 -10806.5} C_VEL
LIN {X 0,Y 557.388,Z 548.955,A -85,B 0,C 180,E1 -10807.764,E2 -10807.764} C_VEL
LIN {X 0,Y 557.782,Z 541.193,A -85,B 0,C 180,E1 -10808.849,E2 -10808.849} C_VEL
LIN {X 0,Y 558.239,Z 531.842,A -85,B 0,C 180,E1 -10809.935,E2 -10809.935} C_VEL
LIN {X 0,Y 558.704,Z 521.426,A -85,B 0,C 180,E1 -10810.931,E2 -10810.931} C_VEL
LIN {X 0,Y 559.358,Z 509.819,A -85,B 0,C 180,E1 -10811.832,E2 -10811.832} C_VEL
LIN {X 0,Y 559.951,Z 497.55,A -85,B 0,C 180,E1 -10812.608,E2 -10812.608} C_VEL
LIN {X 0,Y 560.325,Z 484.355,A -85,B 0,C 180,E1 -10813.279,E2 -10813.279} C_VEL
LIN {X 0,Y 560.621,Z 470.254,A -85,B 0,C 180,E1 -10813.824,E2 -10813.824} C_VEL
LIN {X 0,Y 560.78,Z 456.275,A -85,B 0,C 180,E1 -10814.212,E2 -10814.212} C_VEL
LIN {X 0,Y 561.011,Z 432.463,A -85,B 0,C 180,E1 -10814.622,E2 -10814.622} C_VEL
LIN {X 0,Y 562.712,Z 344.623,A -85,B 0,C 180,E1 -10816.052,E2 -10816.052} C_VEL
LIN {X 0,Y 556.404,Z 329.487,A -85,B 0,C 180,E1 -10816.616,E2 -10816.616} C_VEL
LIN {X 0,Y 556.279,Z 328.754,A -85,B 0,C 180,E1 -10816.636,E2 -10816.636} C_VEL
LIN {X 0,Y 556.244,Z 328.755,A -85,B 0,C 180,E1 -10819.19,E2 -10819.19} C_VEL
LIN {X 0,Y 556.244,Z 328.759,A -85,B 0,C 180,E1 -10822.196,E2 -10822.196} C_VEL
LIN {X 0,Y 556.229,Z 328.755,A -85,B 0,C 180,E1 -10824.949,E2 -10824.949} C_VEL
LIN {X 0,Y 556.253,Z 328.755,A -85,B 0,C 180,E1 -10828.181,E2 -10828.181} C_VEL
LIN {X 0,Y 556.229,Z 328.755,A -85,B 0,C 180,E1 -10831.095,E2 -10831.095} C_VEL
LIN {X 0,Y 556.222,Z 328.756,A -85,B 0,C 180,E1 -10833.784,E2 -10833.784} C_VEL
LIN {X 0,Y 556.259,Z 328.746,A -85,B 0,C 180,E1 -10836.303,E2 -10836.303} C_VEL
LIN {X 0,Y 556.191,Z 328.756,A -85,B 0,C 180,E1 -10839.026,E2 -10839.026} C_VEL
LIN {X 0,Y 556.201,Z 328.752,A -85,B 0,C 180,E1 -10842.011,E2 -10842.011} C_VEL
LIN {X 0,Y 556.25,Z 328.756,A -85,B 0,C 180,E1 -10845.157,E2 -10845.157} C_VEL
LIN {X 0,Y 556.188,Z 328.757,A -85,B 0,C 180,E1 -10848.128,E2 -10848.128} C_VEL
LIN {X 0,Y 556.152,Z 328.768,A -85,B 0,C 180,E1 -10850.97,E2 -10850.97} C_VEL
LIN {X 0,Y 556.214,Z 328.756,A -85,B 0,C 180,E1 -10853.71,E2 -10853.71} C_VEL
LIN {X 0,Y 556.177,Z 328.761,A -85,B 0,C 180,E1 -10856.349,E2 -10856.349} C_VEL
LIN {X 0,Y 556.199,Z 328.763,A -85,B 0,C 180,E1 -10858.913,E2 -10858.913} C_VEL
LIN {X 0,Y 556.235,Z 328.905,A -85,B 0,C 180,E1 -10860.793,E2 -10860.793} C_VEL
LIN {X 0,Y 559.945,Z 345.492,A -85,B 0,C 180,E1 -10862.961,E2 -10862.961} C_VEL
LIN {X 0,Y 560.729,Z 351.229,A -85,B 0,C 180,E1 -10863.675,E2 -10863.675} C_VEL
LIN {X 0,Y 559.654,Z 371.48,A -85,B 0,C 180,E1 -10866.014,E2 -10866.014} C_VEL
LIN {X 0,Y 558.464,Z 396.424,A -85,B 0,C 180,E1 -10868.863,E2 -10868.863} C_VEL
LIN {X 0,Y 557.482,Z 419.739,A -85,B 0,C 180,E1 -10871.503,E2 -10871.503} C_VEL
LIN {X 0,Y 557.214,Z 428.617,A -85,B 0,C 180,E1 -10872.505,E2 -10872.505} C_VEL
LIN {X 0,Y 560.706,Z 457.733,A -85,B 0,C 180,E1 -10873.011,E2 -10873.011} C_VEL
LIN {X 0,Y 561.482,Z 466.391,A -85,B 0,C 180,E1 -10873.15,E2 -10873.15} C_VEL
LIN {X 0,Y 560.392,Z 568.688,A -85,B 0,C 180,E1 -10874.481,E2 -10874.481} C_VEL
LIN {X 0,Y 559.847,Z 583.138,A -85,B 0,C 180,E1 -10874.814,E2 -10874.814} C_VEL
LIN {X 0,Y 559.143,Z 597.612,A -85,B 0,C 180,E1 -10875.305,E2 -10875.305} C_VEL
LIN {X 0,Y 558.378,Z 611.362,A -85,B 0,C 180,E1 -10875.933,E2 -10875.933} C_VEL
LIN {X 0,Y 557.722,Z 623.742,A -85,B 0,C 180,E1 -10876.657,E2 -10876.657} C_VEL
LIN {X 0,Y 556.653,Z 646.304,A -85,B 0,C 180,E1 -10878.201,E2 -10878.201} C_VEL
LIN {X 0,Y 556.242,Z 657.891,A -85,B 0,C 180,E1 -10879.177,E2 -10879.177} C_VEL
LIN {X 0,Y 555.799,Z 667.95,A -85,B 0,C 180,E1 -10880.204,E2 -10880.204} C_VEL
LIN {X 0,Y 555.506,Z 676.805,A -85,B 0,C 180,E1 -10881.297,E2 -10881.297} C_VEL
LIN {X 0,Y 555.225,Z 685.223,A -85,B 0,C 180,E1 -10882.57,E2 -10882.57} C_VEL
LIN {X 0,Y 555.091,Z 691.942,A -85,B 0,C 180,E1 -10883.843,E2 -10883.843} C_VEL
LIN {X 0,Y 555.007,Z 696.575,A -85,B 0,C 180,E1 -10884.932,E2 -10884.932} C_VEL
LIN {X 0,Y 554.939,Z 701.201,A -85,B 0,C 180,E1 -10886.382,E2 -10886.382} C_VEL
LIN {X 0,Y 554.905,Z 704.284,A -85,B 0,C 180,E1 -10887.83,E2 -10887.83} C_VEL
LIN {X 0,Y 554.857,Z 705.91,A -85,B 0,C 180,E1 -10889.277,E2 -10889.277} C_VEL
LIN {X 0,Y 554.856,Z 706.107,A -85,B 0,C 180,E1 -10890.723,E2 -10890.723} C_VEL
LIN {X 0,Y 554.905,Z 704.875,A -85,B 0,C 180,E1 -10892.17,E2 -10892.17} C_VEL
LIN {X 0,Y 554.955,Z 703.71,A -85,B 0,C 180,E1 -10892.894,E2 -10892.894} C_VEL
LIN {X 0,Y 554.972,Z 700.127,A -85,B 0,C 180,E1 -10894.38,E2 -10894.38} C_VEL
LIN {X 0,Y 555.108,Z 695.195,A -85,B 0,C 180,E1 -10895.794,E2 -10895.794} C_VEL
LIN {X 0,Y 555.255,Z 690.294,A -85,B 0,C 180,E1 -10896.883,E2 -10896.883} C_VEL
LIN {X 0,Y 555.549,Z 683.171,A -85,B 0,C 180,E1 -10898.154,E2 -10898.154} C_VEL
LIN {X 0,Y 555.849,Z 675.691,A -85,B 0,C 180,E1 -10899.246,E2 -10899.246} C_VEL
LIN {X 0,Y 556.272,Z 666.782,A -85,B 0,C 180,E1 -10900.325,E2 -10900.325} C_VEL
LIN {X 0,Y 556.71,Z 657.736,A -85,B 0,C 180,E1 -10901.245,E2 -10901.245} C_VEL
LIN {X 0,Y 557.266,Z 645.882,A -85,B 0,C 180,E1 -10902.246,E2 -10902.246} C_VEL
LIN {X 0,Y 557.803,Z 634.02,A -85,B 0,C 180,E1 -10903.063,E2 -10903.063} C_VEL
LIN {X 0,Y 558.42,Z 620.948,A -85,B 0,C 180,E1 -10903.788,E2 -10903.788} C_VEL
LIN {X 0,Y 558.92,Z 607.306,A -85,B 0,C 180,E1 -10904.376,E2 -10904.376} C_VEL
LIN {X 0,Y 559.351,Z 592.393,A -85,B 0,C 180,E1 -10904.852,E2 -10904.852} C_VEL
LIN {X 0,Y 559.729,Z 577.428,A -85,B 0,C 180,E1 -10905.166,E2 -10905.166} C_VEL
LIN {X 0,Y 561.503,Z 484.486,A -85,B 0,C 180,E1 -10906.673,E2 -10906.673} C_VEL
LIN {X 0,Y 561.764,Z 463.063,A -85,B 0,C 180,E1 -10907.046,E2 -10907.046} C_VEL
LIN {X 0,Y 559.552,Z 439.331,A -85,B 0,C 180,E1 -10907.579,E2 -10907.579} C_VEL
LIN {X 0,Y 558.517,Z 430.413,A -85,B 0,C 180,E1 -10907.846,E2 -10907.846} C_VEL
LIN {X 0,Y 557.123,Z 418.326,A -85,B 0,C 180,E1 -10908.293,E2 -10908.293} C_VEL
LIN {X 0,Y 557.893,Z 397.764,A -85,B 0,C 180,E1 -10910.582,E2 -10910.582} C_VEL
LIN {X 0,Y 558.756,Z 375.597,A -85,B 0,C 180,E1 -10913.063,E2 -10913.063} C_VEL
LIN {X 0,Y 559.857,Z 349.862,A -85,B 0,C 180,E1 -10915.969,E2 -10915.969} C_VEL
LIN {X 0,Y 559.791,Z 346.389,A -85,B 0,C 180,E1 -10916.372,E2 -10916.372} C_VEL
LIN {X 0,Y 556.247,Z 328.756,A -85,B 0,C 180,E1 -10918.588,E2 -10918.588} C_VEL
LIN {X 0,Y 556.201,Z 328.759,A -85,B 0,C 180,E1 -10921.091,E2 -10921.091} C_VEL
LIN {X 0,Y 556.176,Z 328.762,A -85,B 0,C 180,E1 -10923.778,E2 -10923.778} C_VEL
LIN {X 0,Y 556.204,Z 328.757,A -85,B 0,C 180,E1 -10926.296,E2 -10926.296} C_VEL
LIN {X 0,Y 556.144,Z 328.767,A -85,B 0,C 180,E1 -10929.03,E2 -10929.03} C_VEL
LIN {X 0,Y 556.195,Z 328.761,A -85,B 0,C 180,E1 -10930.921,E2 -10930.921} C_VEL
LIN {X 0,Y 556.223,Z 328.757,A -85,B 0,C 180,E1 -10934.127,E2 -10934.127} C_VEL
LIN {X 0,Y 556.176,Z 328.763,A -85,B 0,C 180,E1 -10936.924,E2 -10936.924} C_VEL
LIN {X 0,Y 556.18,Z 328.761,A -85,B 0,C 180,E1 -10940.038,E2 -10940.038} C_VEL
LIN {X 0,Y 556.189,Z 328.765,A -85,B 0,C 180,E1 -10942.808,E2 -10942.808} C_VEL
LIN {X 0,Y 556.217,Z 328.759,A -85,B 0,C 180,E1 -10945.481,E2 -10945.481} C_VEL
LIN {X 0,Y 556.204,Z 328.766,A -85,B 0,C 180,E1 -10948.068,E2 -10948.068} C_VEL
LIN {X 0,Y 556.209,Z 328.831,A -85,B 0,C 180,E1 -10950.018,E2 -10950.018} C_VEL
LIN {X 0,Y 560.339,Z 342.607,A -85,B 0,C 180,E1 -10951.843,E2 -10951.843} C_VEL
LIN {X 0,Y 562.748,Z 353.358,A -85,B 0,C 180,E1 -10953.179,E2 -10953.179} C_VEL
LIN {X 0,Y 562.427,Z 366.227,A -85,B 0,C 180,E1 -10954.554,E2 -10954.554} C_VEL
LIN {X 0,Y 561.162,Z 393.688,A -85,B 0,C 180,E1 -10957.469,E2 -10957.469} C_VEL
LIN {X 0,Y 560.072,Z 421.969,A -85,B 0,C 180,E1 -10960.455,E2 -10960.455} C_VEL
LIN {X 0,Y 559.45,Z 439.66,A -85,B 0,C 180,E1 -10962.324,E2 -10962.324} C_VEL
LIN {X 0,Y 562.178,Z 457.715,A -85,B 0,C 180,E1 -10962.776,E2 -10962.776} C_VEL
LIN {X 0,Y 562.536,Z 463.417,A -85,B 0,C 180,E1 -10962.892,E2 -10962.892} C_VEL
LIN {X 0,Y 560.587,Z 558.244,A -85,B 0,C 180,E1 -10964.433,E2 -10964.433} C_VEL
LIN {X 0,Y 560.095,Z 582.594,A -85,B 0,C 180,E1 -10964.844,E2 -10964.844} C_VEL
LIN {X 0,Y 559.639,Z 596.619,A -85,B 0,C 180,E1 -10965.226,E2 -10965.226} C_VEL
LIN {X 0,Y 559.124,Z 609.865,A -85,B 0,C 180,E1 -10965.722,E2 -10965.722} C_VEL
LIN {X 0,Y 558.544,Z 623.775,A -85,B 0,C 180,E1 -10966.401,E2 -10966.401} C_VEL
LIN {X 0,Y 557.84,Z 637.013,A -85,B 0,C 180,E1 -10967.214,E2 -10967.214} C_VEL
LIN {X 0,Y 557.219,Z 648.848,A -85,B 0,C 180,E1 -10968.121,E2 -10968.121} C_VEL
LIN {X 0,Y 556.646,Z 659.588,A -85,B 0,C 180,E1 -10969.12,E2 -10969.12} C_VEL
LIN {X 0,Y 556.218,Z 669.296,A -85,B 0,C 180,E1 -10970.212,E2 -10970.212} C_VEL
LIN {X 0,Y 555.715,Z 677.379,A -85,B 0,C 180,E1 -10971.301,E2 -10971.301} C_VEL
LIN {X 0,Y 555.4,Z 685.111,A -85,B 0,C 180,E1 -10972.573,E2 -10972.573} C_VEL
LIN {X 0,Y 555.161,Z 691.292,A -85,B 0,C 180,E1 -10973.844,E2 -10973.844} C_VEL
LIN {X 0,Y 554.985,Z 695.48,A -85,B 0,C 180,E1 -10974.932,E2 -10974.932} C_VEL
LIN {X 0,Y 554.902,Z 699.69,A -85,B 0,C 180,E1 -10976.382,E2 -10976.382} C_VEL
LIN {X 0,Y 554.847,Z 702.403,A -85,B 0,C 180,E1 -10977.83,E2 -10977.83} C_VEL
LIN {X 0,Y 554.777,Z 703.655,A -85,B 0,C 180,E1 -10979.277,E2 -10979.277} C_VEL
LIN {X 0,Y 554.776,Z 703.493,A -85,B 0,C 180,E1 -10980.724,E2 -10980.724} C_VEL
LIN {X 0,Y 554.845,Z 701.924,A -85,B 0,C 180,E1 -10982.171,E2 -10982.171} C_VEL
LIN {X 0,Y 554.88,Z 698.921,A -85,B 0,C 180,E1 -10983.619,E2 -10983.619} C_VEL
LIN {X 0,Y 554.987,Z 694.409,A -85,B 0,C 180,E1 -10985.069,E2 -10985.069} C_VEL
LIN {X 0,Y 555.076,Z 689.893,A -85,B 0,C 180,E1 -10986.158,E2 -10986.158} C_VEL
LIN {X 0,Y 555.293,Z 683.344,A -85,B 0,C 180,E1 -10987.429,E2 -10987.429} C_VEL
LIN {X 0,Y 555.561,Z 675.18,A -85,B 0,C 180,E1 -10988.702,E2 -10988.702} C_VEL
LIN {X 0,Y 555.94,Z 666.611,A -85,B 0,C 180,E1 -10989.793,E2 -10989.793} C_VEL
LIN {X 0,Y 556.419,Z 655.875,A -85,B 0,C 180,E1 -10990.918,E2 -10990.918} C_VEL
LIN {X 0,Y 556.837,Z 644.647,A -85,B 0,C 180,E1 -10991.887,E2 -10991.887} C_VEL
LIN {X 0,Y 557.337,Z 633.134,A -85,B 0,C 180,E1 -10992.705,E2 -10992.705} C_VEL
LIN {X 0,Y 557.888,Z 620.611,A -85,B 0,C 180,E1 -10993.431,E2 -10993.431} C_VEL
LIN {X 0,Y 558.421,Z 606.683,A -85,B 0,C 180,E1 -10994.065,E2 -10994.065} C_VEL
LIN {X 0,Y 558.745,Z 592.689,A -85,B 0,C 180,E1 -10994.544,E2 -10994.544} C_VEL
LIN {X 0,Y 559.065,Z 578.378,A -85,B 0,C 180,E1 -10994.883,E2 -10994.883} C_VEL
LIN {X 0,Y 560.731,Z 459.87,A -85,B 0,C 180,E1 -10996.664,E2 -10996.664} C_VEL
LIN {X 0,Y 558.224,Z 439.517,A -85,B 0,C 180,E1 -10997.056,E2 -10997.056} C_VEL
LIN {X 0,Y 559.239,Z 408.238,A -85,B 0,C 180,E1 -11000.371,E2 -11000.371} C_VEL
LIN {X 0,Y 560.272,Z 379.89,A -85,B 0,C 180,E1 -11003.387,E2 -11003.387} C_VEL
LIN {X 0,Y 561.243,Z 353.016,A -85,B 0,C 180,E1 -11006.259,E2 -11006.259} C_VEL
LIN {X 0,Y 560.799,Z 348.93,A -85,B 0,C 180,E1 -11006.721,E2 -11006.721} C_VEL
LIN {X 0,Y 556.273,Z 328.755,A -85,B 0,C 180,E1 -11009.102,E2 -11009.102} C_VEL
LIN {X 0,Y 556.225,Z 328.754,A -85,B 0,C 180,E1 -11011.931,E2 -11011.931} C_VEL
LIN {X 0,Y 556.271,Z 328.752,A -85,B 0,C 180,E1 -11015.068,E2 -11015.068} C_VEL
LIN {X 0,Y 556.228,Z 328.756,A -85,B 0,C 180,E1 -11017.501,E2 -11017.501} C_VEL
LIN {X 0,Y 556.2,Z 328.755,A -85,B 0,C 180,E1 -11019.961,E2 -11019.961} C_VEL
LIN {X 0,Y 556.237,Z 328.758,A -85,B 0,C 180,E1 -11023.083,E2 -11023.083} C_VEL
LIN {X 0,Y 556.232,Z 328.751,A -85,B 0,C 180,E1 -11025.872,E2 -11025.872} C_VEL
LIN {X 0,Y 556.209,Z 328.755,A -85,B 0,C 180,E1 -11028.13,E2 -11028.13} C_VEL
LIN {X 0,Y 556.196,Z 328.761,A -85,B 0,C 180,E1 -11030.974,E2 -11030.974} C_VEL
LIN {X 0,Y 556.287,Z 328.745,A -85,B 0,C 180,E1 -11033.715,E2 -11033.715} C_VEL
LIN {X 0,Y 556.223,Z 328.758,A -85,B 0,C 180,E1 -11036.352,E2 -11036.352} C_VEL
LIN {X 0,Y 556.218,Z 328.756,A -85,B 0,C 180,E1 -11038.915,E2 -11038.915} C_VEL
LIN {X 0,Y 556.253,Z 328.751,A -85,B 0,C 180,E1 -11041.819,E2 -11041.819} C_VEL
LIN {X 0,Y 556.208,Z 328.758,A -85,B 0,C 180,E1 -11044.649,E2 -11044.649} C_VEL
LIN {X 0,Y 556.233,Z 328.753,A -85,B 0,C 180,E1 -11047.589,E2 -11047.589} C_VEL
LIN {X 0,Y 555.59,Z 328.84,A -85,B 0,C 180,E1 -11048.193,E2 -11048.193} C_VEL
LIN {X 0,Y 552.762,Z 329.191,A -85,B 0,C 180,E1 -11049.173,E2 -11049.173} C_VEL
LIN {X 0,Y 550.35,Z 329.491,A -85,B 0,C 180,E1 -11049.963,E2 -11049.963} C_VEL
LIN {X 0,Y 549.297,Z 329.618,A -85,B 0,C 180,E1 -11050.572,E2 -11050.572} C_VEL
LIN {X 0,Y 549.204,Z 329.628,A -85,B 0,C 180,E1 -11050.778,E2 -11050.778} C_VEL
LIN {X 0,Y 549.207,Z 329.631,A -85,B 0,C 180,E1 -11053.705,E2 -11053.705} C_VEL
LIN {X 0,Y 549.272,Z 329.626,A -85,B 0,C 180,E1 -11055.978,E2 -11055.978} C_VEL
LIN {X 0,Y 549.276,Z 329.625,A -85,B 0,C 180,E1 -11058.005,E2 -11058.005} C_VEL
LIN {X 0,Y 554.301,Z 344.703,A -85,B 0,C 180,E1 -11058.358,E2 -11058.358} C_VEL
LIN {X 0,Y 553.561,Z 447.862,A -85,B 0,C 180,E1 -11059.704,E2 -11059.704} C_VEL
LIN {X 0,Y 553.432,Z 462.165,A -85,B 0,C 180,E1 -11060.001,E2 -11060.001} C_VEL
LIN {X 0,Y 553.194,Z 475.914,A -85,B 0,C 180,E1 -11060.434,E2 -11060.434} C_VEL
LIN {X 0,Y 552.847,Z 488.722,A -85,B 0,C 180,E1 -11060.98,E2 -11060.98} C_VEL
LIN {X 0,Y 552.414,Z 501.244,A -85,B 0,C 180,E1 -11061.663,E2 -11061.663} C_VEL
LIN {X 0,Y 552.02,Z 512.622,A -85,B 0,C 180,E1 -11062.435,E2 -11062.435} C_VEL
LIN {X 0,Y 551.426,Z 523.675,A -85,B 0,C 180,E1 -11063.344,E2 -11063.344} C_VEL
LIN {X 0,Y 550.852,Z 533.711,A -85,B 0,C 180,E1 -11064.345,E2 -11064.345} C_VEL
LIN {X 0,Y 550.32,Z 542.793,A -85,B 0,C 180,E1 -11065.437,E2 -11065.437} C_VEL
